KUKA KRL program: EPS_2_25694_AC03A_A_20260223033031.src

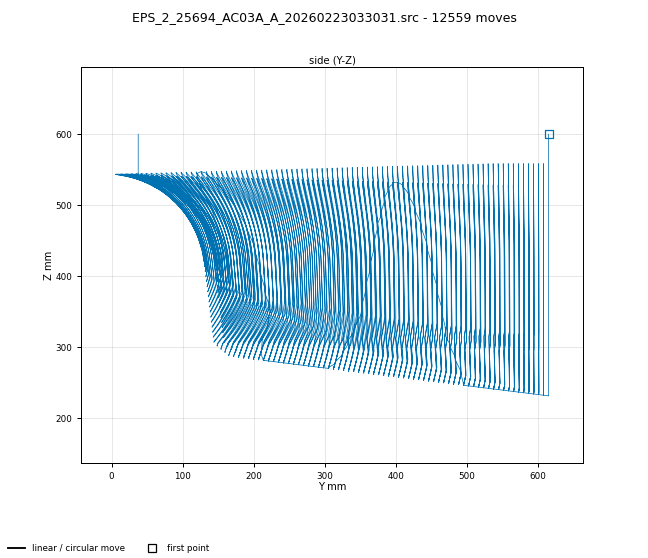
[picture p0: tool path of EPS_2_25694_AC03A_A_20260223033031.src, 12559 of 12561 moves have a stored position in this frame; points joined in program order, loops and branches not executed]
&ACCESS RVP
&REL 4
&COMMENT QRS 19112012
&PARAM EDITMASK = *
DEF PART()
EXT BAS (BAS_COMMAND :IN,REAL :IN )
INT I
BAS (#INITMOV,0 )

;KUKA QRS Post kuka4.cps  Date:22-06-2017 !

File_ID=3050

QRS_PRE_INIT()

;Init var - Until changes are made in qrs_pre_init
Outlet_Square_prg=0
Inlet_1_Square_prg=0
Inlet_2_Square_prg=0
Inlet_3_Square_prg=0
Inlet_4_Square_prg=0
Inlet_5_Square_prg=0

Outlet_1={X 0.000, Y 532.860, Z 433.000, B 0.000, E1 0.000 }
Inlet_1={X 0.000, Y 537.670, Z 428.000, B 0.000, E1 178.000 }
Outlet_1_type=251
Inlet_1_type=201
;QRS#1=Sidecore dimensions
;QRS#2=250-10" PVC SDR 35
;QRS#3=200-8" PVC SDR 35
;QRS#4=
;QRS#5=
;QRS#6=
;QRS#7=
;QRS#8=
;QRS#9=14M PSX
;QRS#10=12-08 PSX
;QRS#11=
;QRS#12=
;QRS#13=
;QRS#14=
;QRS#15=
;QRS#16=1220x127x838 2,75'
;QRS#17=EPS Height
;QRS#18=558,5
;QRS#19=*
;QRS#20= UPDATED VERSION 22-06-2017
;QRS#21=*
Outlet_Square=0100
Inlet_1_Square=0100
Inlet_2_Square=0
Inlet_3_Square=0
Inlet_4_Square=0
Inlet_5_Square=0
Mill_Square=1
Outlet_Square_Prg=205
Inlet_1_Square_prg=204

QRS_INIT()

$ADVANCE=5

; T1
PTP {E1 173.602,E2 173.602}
PTP {X 0,Y 615.5,A -85,B 0,C 180,E1 173.602,E2 173.602,E3 0,E4 0,E5 0,E6 0}
QRS_SPEED_INIT()
LIN {X 0,Y 615.5,Z 600,A -85,B 0,C 180,E1 173.602,E2 173.602,E3 0,E4 0,E5 0,E6 0} C_VEL
LIN {X 0,Y 615.5,Z 241.488,A -85,B 0,C 180,E1 173.602,E2 173.602} C_VEL
LIN {X 0,Y 615.5,Z 233.308,A -85,B 0,C 180,E1 173.602,E2 173.602} C_VEL
LIN {X 0,Y 615.485,Z 231.308,A -85,B 0,C 180,E1 173.415,E2 173.415} C_VEL
LIN {X 0,Y 615.485,Z 231.321,A -85,B 0,C 180,E1 170.801,E2 170.801} C_VEL
LIN {X 0,Y 615.479,Z 231.314,A -85,B 0,C 180,E1 168.139,E2 168.139} C_VEL
LIN {X 0,Y 615.48,Z 231.31,A -85,B 0,C 180,E1 165.45,E2 165.45} C_VEL
LIN {X 0,Y 615.496,Z 231.326,A -85,B 0,C 180,E1 162.729,E2 162.729} C_VEL
LIN {X 0,Y 615.49,Z 231.307,A -85,B 0,C 180,E1 159.967,E2 159.967} C_VEL
LIN {X 0,Y 615.477,Z 231.319,A -85,B 0,C 180,E1 157.155,E2 157.155} C_VEL
LIN {X 0,Y 615.48,Z 231.316,A -85,B 0,C 180,E1 154.431,E2 154.431} C_VEL
LIN {X 0,Y 615.484,Z 231.309,A -85,B 0,C 180,E1 152.084,E2 152.084} C_VEL
LIN {X 0,Y 615.487,Z 231.308,A -85,B 0,C 180,E1 149.839,E2 149.839} C_VEL
LIN {X 0,Y 615.475,Z 231.314,A -85,B 0,C 180,E1 147.541,E2 147.541} C_VEL
LIN {X 0,Y 615.486,Z 231.322,A -85,B 0,C 180,E1 145.184,E2 145.184} C_VEL
LIN {X 0,Y 615.483,Z 231.319,A -85,B 0,C 180,E1 142.757,E2 142.757} C_VEL
LIN {X 0,Y 615.481,Z 231.31,A -85,B 0,C 180,E1 139.911,E2 139.911} C_VEL
LIN {X 0,Y 615.475,Z 231.315,A -85,B 0,C 180,E1 137.645,E2 137.645} C_VEL
LIN {X 0,Y 615.484,Z 231.32,A -85,B 0,C 180,E1 134.931,E2 134.931} C_VEL
LIN {X 0,Y 615.483,Z 231.309,A -85,B 0,C 180,E1 132.079,E2 132.079} C_VEL
LIN {X 0,Y 615.475,Z 231.316,A -85,B 0,C 180,E1 129.75,E2 129.75} C_VEL
LIN {X 0,Y 615.481,Z 231.317,A -85,B 0,C 180,E1 126.935,E2 126.935} C_VEL
LIN {X 0,Y 615.484,Z 231.311,A -85,B 0,C 180,E1 124.699,E2 124.699} C_VEL
LIN {X 0,Y 615.489,Z 231.307,A -85,B 0,C 180,E1 122.33,E2 122.33} C_VEL
LIN {X 0,Y 615.492,Z 231.326,A -85,B 0,C 180,E1 119.406,E2 119.406} C_VEL
LIN {X 0,Y 615.485,Z 231.308,A -85,B 0,C 180,E1 116.444,E2 116.444} C_VEL
LIN {X 0,Y 615.496,Z 231.499,A -85,B 0,C 180,E1 115.424,E2 115.424} C_VEL
LIN {X 0,Y 615.497,Z 234.472,A -85,B 0,C 180,E1 114.991,E2 114.991} C_VEL
LIN {X 0,Y 615.466,Z 256.829,A -85,B 0,C 180,E1 112.137,E2 112.137} C_VEL
LIN {X 0,Y 615.461,Z 277.73,A -85,B 0,C 180,E1 109.512,E2 109.512} C_VEL
LIN {X 0,Y 615.491,Z 299.956,A -85,B 0,C 180,E1 106.757,E2 106.757} C_VEL
LIN {X 0,Y 615.493,Z 315.536,A -85,B 0,C 180,E1 104.866,E2 104.866} C_VEL
LIN {X 0,Y 615.498,Z 318.146,A -85,B 0,C 180,E1 104.802,E2 104.802} C_VEL
LIN {X 0,Y 615.5,Z 424.718,A -85,B 0,C 180,E1 103.537,E2 103.537} C_VEL
LIN {X 0,Y 615.499,Z 437.939,A -85,B 0,C 180,E1 103.243,E2 103.243} C_VEL
LIN {X 0,Y 615.498,Z 450.618,A -85,B 0,C 180,E1 102.823,E2 102.823} C_VEL
LIN {X 0,Y 615.485,Z 462.672,A -85,B 0,C 180,E1 102.279,E2 102.279} C_VEL
LIN {X 0,Y 615.496,Z 474.125,A -85,B 0,C 180,E1 101.61,E2 101.61} C_VEL
LIN {X 0,Y 615.496,Z 484.042,A -85,B 0,C 180,E1 100.889,E2 100.889} C_VEL
LIN {X 0,Y 615.497,Z 493.658,A -85,B 0,C 180,E1 100.028,E2 100.028} C_VEL
LIN {X 0,Y 615.496,Z 502.594,A -85,B 0,C 180,E1 99.033,E2 99.033} C_VEL
LIN {X 0,Y 615.497,Z 509.771,A -85,B 0,C 180,E1 98.041,E2 98.041} C_VEL
LIN {X 0,Y 615.496,Z 516.224,A -85,B 0,C 180,E1 96.898,E2 96.898} C_VEL
LIN {X 0,Y 615.499,Z 520.584,A -85,B 0,C 180,E1 95.898,E2 95.898} C_VEL
LIN {X 0,Y 615.498,Z 522.856,A -85,B 0,C 180,E1 95.241,E2 95.241} C_VEL
LIN {X 0,Y 615.496,Z 524.703,A -85,B 0,C 180,E1 94.584,E2 94.584} C_VEL
LIN {X 0,Y 615.496,Z 526.091,A -85,B 0,C 180,E1 93.928,E2 93.928} C_VEL
LIN {X 0,Y 615.495,Z 527.668,A -85,B 0,C 180,E1 92.618,E2 92.618} C_VEL
LIN {X 0,Y 615.5,Z 527.887,A -85,B 0,C 180,E1 91.963,E2 91.963} C_VEL
LIN {X 0,Y 615.495,Z 527.089,A -85,B 0,C 180,E1 90.654,E2 90.654} C_VEL
LIN {X 0,Y 615.497,Z 526.122,A -85,B 0,C 180,E1 90,E2 90} C_VEL
LIN {X 0,Y 615.494,Z 524.755,A -85,B 0,C 180,E1 89.346,E2 89.346} C_VEL
LIN {X 0,Y 615.496,Z 521.882,A -85,B 0,C 180,E1 88.364,E2 88.364} C_VEL
LIN {X 0,Y 615.498,Z 517.992,A -85,B 0,C 180,E1 87.382,E2 87.382} C_VEL
LIN {X 0,Y 615.496,Z 512.983,A -85,B 0,C 180,E1 86.399,E2 86.399} C_VEL
LIN {X 0,Y 615.498,Z 506.694,A -85,B 0,C 180,E1 85.416,E2 85.416} C_VEL
LIN {X 0,Y 615.498,Z 498.82,A -85,B 0,C 180,E1 84.43,E2 84.43} C_VEL
LIN {X 0,Y 615.498,Z 489.04,A -85,B 0,C 180,E1 83.444,E2 83.444} C_VEL
LIN {X 0,Y 615.499,Z 478.771,A -85,B 0,C 180,E1 82.62,E2 82.62} C_VEL
LIN {X 0,Y 615.488,Z 467.229,A -85,B 0,C 180,E1 81.877,E2 81.877} C_VEL
LIN {X 0,Y 615.497,Z 455.695,A -85,B 0,C 180,E1 81.298,E2 81.298} C_VEL
LIN {X 0,Y 615.498,Z 443.77,A -85,B 0,C 180,E1 80.843,E2 80.843} C_VEL
LIN {X 0,Y 615.499,Z 431.72,A -85,B 0,C 180,E1 80.512,E2 80.512} C_VEL
LIN {X 0,Y 615.497,Z 418.522,A -85,B 0,C 180,E1 80.283,E2 80.283} C_VEL
LIN {X 0,Y 615.49,Z 316.121,A -85,B 0,C 180,E1 79.075,E2 79.075} C_VEL
LIN {X 0,Y 615.49,Z 314.695,A -85,B 0,C 180,E1 78.96,E2 78.96} C_VEL
LIN {X 0,Y 615.492,Z 291.637,A -85,B 0,C 180,E1 76.126,E2 76.126} C_VEL
LIN {X 0,Y 615.485,Z 267.127,A -85,B 0,C 180,E1 73.072,E2 73.072} C_VEL
LIN {X 0,Y 615.462,Z 245.356,A -85,B 0,C 180,E1 70.315,E2 70.315} C_VEL
LIN {X 0,Y 615.495,Z 231.626,A -85,B 0,C 180,E1 68.525,E2 68.525} C_VEL
LIN {X 0,Y 615.481,Z 231.31,A -85,B 0,C 180,E1 67.657,E2 67.657} C_VEL
LIN {X 0,Y 615.478,Z 231.314,A -85,B 0,C 180,E1 65.008,E2 65.008} C_VEL
LIN {X 0,Y 615.482,Z 231.318,A -85,B 0,C 180,E1 62.823,E2 62.823} C_VEL
LIN {X 0,Y 615.477,Z 231.319,A -85,B 0,C 180,E1 60.208,E2 60.208} C_VEL
LIN {X 0,Y 615.493,Z 231.306,A -85,B 0,C 180,E1 57.544,E2 57.544} C_VEL
LIN {X 0,Y 615.48,Z 231.313,A -85,B 0,C 180,E1 55.185,E2 55.185} C_VEL
LIN {X 0,Y 615.485,Z 231.325,A -85,B 0,C 180,E1 52.758,E2 52.758} C_VEL
LIN {X 0,Y 615.48,Z 231.31,A -85,B 0,C 180,E1 49.913,E2 49.913} C_VEL
LIN {X 0,Y 615.496,Z 231.306,A -85,B 0,C 180,E1 47.649,E2 47.649} C_VEL
LIN {X 0,Y 615.486,Z 231.323,A -85,B 0,C 180,E1 44.932,E2 44.932} C_VEL
LIN {X 0,Y 615.481,Z 231.31,A -85,B 0,C 180,E1 42.081,E2 42.081} C_VEL
LIN {X 0,Y 615.49,Z 231.307,A -85,B 0,C 180,E1 39.75,E2 39.75} C_VEL
LIN {X 0,Y 615.486,Z 231.328,A -85,B 0,C 180,E1 36.938,E2 36.938} C_VEL
LIN {X 0,Y 615.487,Z 231.308,A -85,B 0,C 180,E1 34.022,E2 34.022} C_VEL
LIN {X 0,Y 615.482,Z 231.327,A -85,B 0,C 180,E1 31.087,E2 31.087} C_VEL
LIN {X 0,Y 615.477,Z 231.313,A -85,B 0,C 180,E1 28.45,E2 28.45} C_VEL
LIN {X 0,Y 615.481,Z 231.312,A -85,B 0,C 180,E1 25.716,E2 25.716} C_VEL
LIN {X 0,Y 615.478,Z 231.317,A -85,B 0,C 180,E1 23.557,E2 23.557} C_VEL
LIN {X 0,Y 615.483,Z 231.32,A -85,B 0,C 180,E1 21.432,E2 21.432} C_VEL
LIN {X 0,Y 615.476,Z 231.313,A -85,B 0,C 180,E1 18.605,E2 18.605} C_VEL
LIN {X 0,Y 615.478,Z 231.312,A -85,B 0,C 180,E1 15.906,E2 15.906} C_VEL
LIN {X 0,Y 615.491,Z 231.323,A -85,B 0,C 180,E1 13.201,E2 13.201} C_VEL
LIN {X 0,Y 615.485,Z 231.309,A -85,B 0,C 180,E1 10.527,E2 10.527} C_VEL
LIN {X 0,Y 615.479,Z 231.315,A -85,B 0,C 180,E1 7.876,E2 7.876} C_VEL
LIN {X 0,Y 615.485,Z 231.321,A -85,B 0,C 180,E1 5.241,E2 5.241} C_VEL
LIN {X 0,Y 615.487,Z 231.308,A -85,B 0,C 180,E1 2.618,E2 2.618} C_VEL
LIN {X 0,Y 615.479,Z 231.315,A -85,B 0,C 180,E1 0,E2 0} C_VEL
LIN {X 0,Y 615.485,Z 231.321,A -85,B 0,C 180,E1 -2.618,E2 -2.618} C_VEL
LIN {X 0,Y 615.487,Z 231.308,A -85,B 0,C 180,E1 -5.241,E2 -5.241} C_VEL
LIN {X 0,Y 615.479,Z 231.315,A -85,B 0,C 180,E1 -7.876,E2 -7.876} C_VEL
LIN {X 0,Y 615.484,Z 231.321,A -85,B 0,C 180,E1 -10.527,E2 -10.527} C_VEL
LIN {X 0,Y 615.493,Z 231.306,A -85,B 0,C 180,E1 -13.201,E2 -13.201} C_VEL
LIN {X 0,Y 615.482,Z 231.319,A -85,B 0,C 180,E1 -15.905,E2 -15.905} C_VEL
LIN {X 0,Y 615.475,Z 231.316,A -85,B 0,C 180,E1 -18.646,E2 -18.646} C_VEL
LIN {X 0,Y 615.479,Z 231.311,A -85,B 0,C 180,E1 -21.432,E2 -21.432} C_VEL
LIN {X 0,Y 615.483,Z 231.322,A -85,B 0,C 180,E1 -24.272,E2 -24.272} C_VEL
LIN {X 0,Y 615.49,Z 231.307,A -85,B 0,C 180,E1 -27.177,E2 -27.177} C_VEL
LIN {X 0,Y 615.486,Z 231.321,A -85,B 0,C 180,E1 -30.16,E2 -30.16} C_VEL
LIN {X 0,Y 615.472,Z 231.316,A -85,B 0,C 180,E1 -32.458,E2 -32.458} C_VEL
LIN {X 0,Y 615.49,Z 231.307,A -85,B 0,C 180,E1 -34.815,E2 -34.815} C_VEL
LIN {X 0,Y 615.48,Z 231.312,A -85,B 0,C 180,E1 -37.243,E2 -37.243} C_VEL
LIN {X 0,Y 615.482,Z 231.32,A -85,B 0,C 180,E1 -40.09,E2 -40.09} C_VEL
LIN {X 0,Y 615.476,Z 231.314,A -85,B 0,C 180,E1 -42.354,E2 -42.354} C_VEL
LIN {X 0,Y 615.481,Z 231.311,A -85,B 0,C 180,E1 -45.069,E2 -45.069} C_VEL
LIN {X 0,Y 615.484,Z 231.32,A -85,B 0,C 180,E1 -47.92,E2 -47.92} C_VEL
LIN {X 0,Y 615.477,Z 231.313,A -85,B 0,C 180,E1 -50.25,E2 -50.25} C_VEL
LIN {X 0,Y 615.476,Z 231.314,A -85,B 0,C 180,E1 -53.065,E2 -53.065} C_VEL
LIN {X 0,Y 615.482,Z 231.32,A -85,B 0,C 180,E1 -55.3,E2 -55.3} C_VEL
LIN {X 0,Y 615.489,Z 231.322,A -85,B 0,C 180,E1 -57.669,E2 -57.669} C_VEL
LIN {X 0,Y 615.492,Z 231.307,A -85,B 0,C 180,E1 -60.595,E2 -60.595} C_VEL
LIN {X 0,Y 615.485,Z 231.324,A -85,B 0,C 180,E1 -63.556,E2 -63.556} C_VEL
LIN {X 0,Y 615.485,Z 231.308,A -85,B 0,C 180,E1 -66.444,E2 -66.444} C_VEL
LIN {X 0,Y 615.499,Z 231.499,A -85,B 0,C 180,E1 -67.466,E2 -67.466} C_VEL
LIN {X 0,Y 615.496,Z 239.528,A -85,B 0,C 180,E1 -68.393,E2 -68.393} C_VEL
LIN {X 0,Y 615.453,Z 264.946,A -85,B 0,C 180,E1 -71.181,E2 -71.181} C_VEL
LIN {X 0,Y 615.44,Z 287.175,A -85,B 0,C 180,E1 -73.584,E2 -73.584} C_VEL
LIN {X 0,Y 615.491,Z 294.635,A -85,B 0,C 180,E1 -74.371,E2 -74.371} C_VEL
LIN {X 0,Y 615.486,Z 299.642,A -85,B 0,C 180,E1 -74.456,E2 -74.456} C_VEL
LIN {X 0,Y 615.499,Z 433.907,A -85,B 0,C 180,E1 -76.063,E2 -76.063} C_VEL
LIN {X 0,Y 615.497,Z 448.387,A -85,B 0,C 180,E1 -76.379,E2 -76.379} C_VEL
LIN {X 0,Y 615.495,Z 461.695,A -85,B 0,C 180,E1 -76.799,E2 -76.799} C_VEL
LIN {X 0,Y 615.497,Z 473.842,A -85,B 0,C 180,E1 -77.303,E2 -77.303} C_VEL
LIN {X 0,Y 615.484,Z 486.604,A -85,B 0,C 180,E1 -77.972,E2 -77.972} C_VEL
LIN {X 0,Y 615.499,Z 499.343,A -85,B 0,C 180,E1 -78.807,E2 -78.807} C_VEL
LIN {X 0,Y 615.498,Z 509.751,A -85,B 0,C 180,E1 -79.64,E2 -79.64} C_VEL
LIN {X 0,Y 615.496,Z 520.09,A -85,B 0,C 180,E1 -80.636,E2 -80.636} C_VEL
LIN {X 0,Y 615.497,Z 528.604,A -85,B 0,C 180,E1 -81.629,E2 -81.629} C_VEL
LIN {X 0,Y 615.496,Z 536.728,A -85,B 0,C 180,E1 -82.785,E2 -82.785} C_VEL
LIN {X 0,Y 615.497,Z 542.431,A -85,B 0,C 180,E1 -83.773,E2 -83.773} C_VEL
LIN {X 0,Y 615.495,Z 547.081,A -85,B 0,C 180,E1 -84.759,E2 -84.759} C_VEL
LIN {X 0,Y 615.494,Z 551.902,A -85,B 0,C 180,E1 -86.072,E2 -86.072} C_VEL
LIN {X 0,Y 615.496,Z 555.252,A -85,B 0,C 180,E1 -87.382,E2 -87.382} C_VEL
LIN {X 0,Y 615.489,Z 557.229,A -85,B 0,C 180,E1 -88.691,E2 -88.691} C_VEL
LIN {X 0,Y 615.493,Z 557.889,A -85,B 0,C 180,E1 -90,E2 -90} C_VEL
LIN {X 0,Y 615.489,Z 557.229,A -85,B 0,C 180,E1 -91.309,E2 -91.309} C_VEL
LIN {X 0,Y 615.496,Z 555.252,A -85,B 0,C 180,E1 -92.618,E2 -92.618} C_VEL
LIN {X 0,Y 615.494,Z 551.902,A -85,B 0,C 180,E1 -93.928,E2 -93.928} C_VEL
LIN {X 0,Y 615.495,Z 547.08,A -85,B 0,C 180,E1 -95.241,E2 -95.241} C_VEL
LIN {X 0,Y 615.496,Z 540.628,A -85,B 0,C 180,E1 -96.556,E2 -96.556} C_VEL
LIN {X 0,Y 615.496,Z 533.441,A -85,B 0,C 180,E1 -97.71,E2 -97.71} C_VEL
LIN {X 0,Y 615.498,Z 525.904,A -85,B 0,C 180,E1 -98.702,E2 -98.702} C_VEL
LIN {X 0,Y 615.496,Z 516.854,A -85,B 0,C 180,E1 -99.696,E2 -99.696} C_VEL
LIN {X 0,Y 615.498,Z 506.758,A -85,B 0,C 180,E1 -100.618,E2 -100.618} C_VEL
LIN {X 0,Y 615.498,Z 495.859,A -85,B 0,C 180,E1 -101.443,E2 -101.443} C_VEL
LIN {X 0,Y 615.485,Z 483.709,A -85,B 0,C 180,E1 -102.195,E2 -102.195} C_VEL
LIN {X 0,Y 615.494,Z 470.094,A -85,B 0,C 180,E1 -102.865,E2 -102.865} C_VEL
LIN {X 0,Y 615.495,Z 456.839,A -85,B 0,C 180,E1 -103.369,E2 -103.369} C_VEL
LIN {X 0,Y 615.498,Z 443.293,A -85,B 0,C 180,E1 -103.747,E2 -103.747} C_VEL
LIN {X 0,Y 615.498,Z 428.744,A -85,B 0,C 180,E1 -104.013,E2 -104.013} C_VEL
LIN {X 0,Y 615.49,Z 295.04,A -85,B 0,C 180,E1 -105.607,E2 -105.607} C_VEL
LIN {X 0,Y 615.462,Z 289.547,A -85,B 0,C 180,E1 -106.16,E2 -106.16} C_VEL
LIN {X 0,Y 615.445,Z 266.533,A -85,B 0,C 180,E1 -108.647,E2 -108.647} C_VEL
LIN {X 0,Y 615.499,Z 241.116,A -85,B 0,C 180,E1 -111.431,E2 -111.431} C_VEL
LIN {X 0,Y 615.499,Z 231.618,A -85,B 0,C 180,E1 -112.503,E2 -112.503} C_VEL
LIN {X 0,Y 615.483,Z 231.321,A -85,B 0,C 180,E1 -112.844,E2 -112.844} C_VEL
LIN {X 0,Y 615.486,Z 231.308,A -85,B 0,C 180,E1 -115.715,E2 -115.715} C_VEL
LIN {X 0,Y 615.484,Z 231.324,A -85,B 0,C 180,E1 -118.658,E2 -118.658} C_VEL
LIN {X 0,Y 615.479,Z 231.313,A -85,B 0,C 180,E1 -121.085,E2 -121.085} C_VEL
LIN {X 0,Y 615.492,Z 231.306,A -85,B 0,C 180,E1 -123.535,E2 -123.535} C_VEL
LIN {X 0,Y 615.484,Z 231.328,A -85,B 0,C 180,E1 -126.424,E2 -126.424} C_VEL
LIN {X 0,Y 615.482,Z 231.311,A -85,B 0,C 180,E1 -129.061,E2 -129.061} C_VEL
LIN {X 0,Y 615.486,Z 231.308,A -85,B 0,C 180,E1 -131.473,E2 -131.473} C_VEL
LIN {X 0,Y 615.489,Z 231.322,A -85,B 0,C 180,E1 -134.148,E2 -134.148} C_VEL
LIN {X 0,Y 615.482,Z 231.31,A -85,B 0,C 180,E1 -136.952,E2 -136.952} C_VEL
LIN {X 0,Y 615.481,Z 231.31,A -85,B 0,C 180,E1 -139.393,E2 -139.393} C_VEL
LIN {X 0,Y 615.48,Z 231.323,A -85,B 0,C 180,E1 -141.988,E2 -141.988} C_VEL
LIN {X 0,Y 615.479,Z 231.32,A -85,B 0,C 180,E1 -144.384,E2 -144.384} C_VEL
LIN {X 0,Y 615.482,Z 231.311,A -85,B 0,C 180,E1 -146.764,E2 -146.764} C_VEL
LIN {X 0,Y 615.487,Z 231.308,A -85,B 0,C 180,E1 -149.08,E2 -149.08} C_VEL
LIN {X 0,Y 615.477,Z 231.316,A -85,B 0,C 180,E1 -151.55,E2 -151.55} C_VEL
LIN {X 0,Y 615.477,Z 231.319,A -85,B 0,C 180,E1 -154.284,E2 -154.284} C_VEL
LIN {X 0,Y 615.477,Z 231.315,A -85,B 0,C 180,E1 -156.443,E2 -156.443} C_VEL
LIN {X 0,Y 615.479,Z 231.311,A -85,B 0,C 180,E1 -158.568,E2 -158.568} C_VEL
LIN {X 0,Y 615.475,Z 231.316,A -85,B 0,C 180,E1 -161.396,E2 -161.396} C_VEL
LIN {X 0,Y 615.482,Z 231.319,A -85,B 0,C 180,E1 -164.095,E2 -164.095} C_VEL
LIN {X 0,Y 615.493,Z 231.306,A -85,B 0,C 180,E1 -166.799,E2 -166.799} C_VEL
LIN {X 0,Y 615.483,Z 231.32,A -85,B 0,C 180,E1 -169.473,E2 -169.473} C_VEL
LIN {X 0,Y 615.479,Z 231.315,A -85,B 0,C 180,E1 -172.124,E2 -172.124} C_VEL
LIN {X 0,Y 615.487,Z 231.308,A -85,B 0,C 180,E1 -174.759,E2 -174.759} C_VEL
LIN {X 0,Y 615.485,Z 231.321,A -85,B 0,C 180,E1 -177.382,E2 -177.382} C_VEL
LIN {X 0,Y 615.479,Z 231.315,A -85,B 0,C 180,E1 -180,E2 -180} C_VEL
LIN {X 0,Y 615.487,Z 231.308,A -85,B 0,C 180,E1 -182.618,E2 -182.618} C_VEL
LIN {X 0,Y 615.484,Z 231.321,A -85,B 0,C 180,E1 -185.241,E2 -185.241} C_VEL
LIN {X 0,Y 615.485,Z 231.308,A -85,B 0,C 180,E1 -186.585,E2 -186.585} C_VEL
LIN {X 0,Y 614.809,Z 231.468,A -85,B 0,C 180,E1 -187.131,E2 -187.131} C_VEL
LIN {X 0,Y 611.975,Z 231.875,A -85,B 0,C 180,E1 -188.017,E2 -188.017} C_VEL
LIN {X 0,Y 609.583,Z 232.191,A -85,B 0,C 180,E1 -188.729,E2 -188.729} C_VEL
LIN {X 0,Y 608.546,Z 232.311,A -85,B 0,C 180,E1 -189.279,E2 -189.279} C_VEL
LIN {X 0,Y 608.456,Z 232.318,A -85,B 0,C 180,E1 -189.465,E2 -189.465} C_VEL
LIN {X 0,Y 608.455,Z 232.313,A -85,B 0,C 180,E1 -192,E2 -192} C_VEL
LIN {X 0,Y 608.47,Z 232.312,A -85,B 0,C 180,E1 -194.721,E2 -194.721} C_VEL
LIN {X 0,Y 608.457,Z 232.319,A -85,B 0,C 180,E1 -197.477,E2 -197.477} C_VEL
LIN {X 0,Y 608.46,Z 232.311,A -85,B 0,C 180,E1 -200.275,E2 -200.275} C_VEL
LIN {X 0,Y 608.452,Z 232.313,A -85,B 0,C 180,E1 -202.477,E2 -202.477} C_VEL
LIN {X 0,Y 608.453,Z 232.314,A -85,B 0,C 180,E1 -204.571,E2 -204.571} C_VEL
LIN {X 0,Y 608.482,Z 232.317,A -85,B 0,C 180,E1 -207.21,E2 -207.21} C_VEL
LIN {X 0,Y 608.467,Z 232.31,A -85,B 0,C 180,E1 -209.973,E2 -209.973} C_VEL
LIN {X 0,Y 608.451,Z 232.315,A -85,B 0,C 180,E1 -212.522,E2 -212.522} C_VEL
LIN {X 0,Y 608.441,Z 232.319,A -85,B 0,C 180,E1 -215.278,E2 -215.278} C_VEL
LIN {X 0,Y 608.466,Z 232.311,A -85,B 0,C 180,E1 -217.747,E2 -217.747} C_VEL
LIN {X 0,Y 608.445,Z 232.315,A -85,B 0,C 180,E1 -220.329,E2 -220.329} C_VEL
LIN {X 0,Y 608.452,Z 232.321,A -85,B 0,C 180,E1 -222.961,E2 -222.961} C_VEL
LIN {X 0,Y 608.459,Z 232.312,A -85,B 0,C 180,E1 -225.737,E2 -225.737} C_VEL
LIN {X 0,Y 608.46,Z 232.32,A -85,B 0,C 180,E1 -228.659,E2 -228.659} C_VEL
LIN {X 0,Y 608.462,Z 232.311,A -85,B 0,C 180,E1 -231.761,E2 -231.761} C_VEL
LIN {X 0,Y 608.445,Z 232.314,A -85,B 0,C 180,E1 -233.956,E2 -233.956} C_VEL
LIN {X 0,Y 608.446,Z 232.318,A -85,B 0,C 180,E1 -236.329,E2 -236.329} C_VEL
LIN {X 0,Y 608.448,Z 232.321,A -85,B 0,C 180,E1 -238.733,E2 -238.733} C_VEL
LIN {X 0,Y 608.474,Z 232.31,A -85,B 0,C 180,E1 -241.381,E2 -241.381} C_VEL
LIN {X 0,Y 608.473,Z 232.318,A -85,B 0,C 180,E1 -244.28,E2 -244.28} C_VEL
LIN {X 0,Y 608.531,Z 232.698,A -85,B 0,C 180,E1 -244.484,E2 -244.484} C_VEL
LIN {X 0,Y 608.565,Z 248.251,A -85,B 0,C 180,E1 -246.521,E2 -246.521} C_VEL
LIN {X 0,Y 608.534,Z 270.042,A -85,B 0,C 180,E1 -249.306,E2 -249.306} C_VEL
LIN {X 0,Y 608.506,Z 292.884,A -85,B 0,C 180,E1 -252.178,E2 -252.178} C_VEL
LIN {X 0,Y 608.484,Z 315.353,A -85,B 0,C 180,E1 -254.959,E2 -254.959} C_VEL
LIN {X 0,Y 608.564,Z 316.492,A -85,B 0,C 180,E1 -255.025,E2 -255.025} C_VEL
LIN {X 0,Y 608.551,Z 424.72,A -85,B 0,C 180,E1 -256.327,E2 -256.327} C_VEL
LIN {X 0,Y 608.548,Z 437.979,A -85,B 0,C 180,E1 -256.624,E2 -256.624} C_VEL
LIN {X 0,Y 608.527,Z 450.13,A -85,B 0,C 180,E1 -257.027,E2 -257.027} C_VEL
LIN {X 0,Y 608.491,Z 462.397,A -85,B 0,C 180,E1 -257.578,E2 -257.578} C_VEL
LIN {X 0,Y 608.501,Z 473.977,A -85,B 0,C 180,E1 -258.255,E2 -258.255} C_VEL
LIN {X 0,Y 608.481,Z 484.737,A -85,B 0,C 180,E1 -259.042,E2 -259.042} C_VEL
LIN {X 0,Y 608.482,Z 493.745,A -85,B 0,C 180,E1 -259.855,E2 -259.855} C_VEL
LIN {X 0,Y 608.47,Z 502.779,A -85,B 0,C 180,E1 -260.862,E2 -260.862} C_VEL
LIN {X 0,Y 608.463,Z 510.05,A -85,B 0,C 180,E1 -261.866,E2 -261.866} C_VEL
LIN {X 0,Y 608.445,Z 514.948,A -85,B 0,C 180,E1 -262.7,E2 -262.7} C_VEL
LIN {X 0,Y 608.452,Z 519.411,A -85,B 0,C 180,E1 -263.632,E2 -263.632} C_VEL
LIN {X 0,Y 608.442,Z 523.341,A -85,B 0,C 180,E1 -264.698,E2 -264.698} C_VEL
LIN {X 0,Y 608.429,Z 525.219,A -85,B 0,C 180,E1 -265.362,E2 -265.362} C_VEL
LIN {X 0,Y 608.433,Z 526.646,A -85,B 0,C 180,E1 -266.026,E2 -266.026} C_VEL
LIN {X 0,Y 608.421,Z 528.261,A -85,B 0,C 180,E1 -267.352,E2 -267.352} C_VEL
LIN {X 0,Y 608.445,Z 528.498,A -85,B 0,C 180,E1 -268.014,E2 -268.014} C_VEL
LIN {X 0,Y 608.447,Z 528.305,A -85,B 0,C 180,E1 -268.676,E2 -268.676} C_VEL
LIN {X 0,Y 608.437,Z 526.753,A -85,B 0,C 180,E1 -270,E2 -270} C_VEL
LIN {X 0,Y 608.437,Z 525.387,A -85,B 0,C 180,E1 -270.662,E2 -270.662} C_VEL
LIN {X 0,Y 608.44,Z 522.503,A -85,B 0,C 180,E1 -271.655,E2 -271.655} C_VEL
LIN {X 0,Y 608.432,Z 518.599,A -85,B 0,C 180,E1 -272.648,E2 -272.648} C_VEL
LIN {X 0,Y 608.449,Z 513.569,A -85,B 0,C 180,E1 -273.642,E2 -273.642} C_VEL
LIN {X 0,Y 608.465,Z 507.261,A -85,B 0,C 180,E1 -274.637,E2 -274.637} C_VEL
LIN {X 0,Y 608.47,Z 499.369,A -85,B 0,C 180,E1 -275.634,E2 -275.634} C_VEL
LIN {X 0,Y 608.485,Z 489.571,A -85,B 0,C 180,E1 -276.632,E2 -276.632} C_VEL
LIN {X 0,Y 608.479,Z 479.318,A -85,B 0,C 180,E1 -277.466,E2 -277.466} C_VEL
LIN {X 0,Y 608.505,Z 467.794,A -85,B 0,C 180,E1 -278.217,E2 -278.217} C_VEL
LIN {X 0,Y 608.519,Z 456.378,A -85,B 0,C 180,E1 -278.802,E2 -278.802} C_VEL
LIN {X 0,Y 608.547,Z 444.602,A -85,B 0,C 180,E1 -279.263,E2 -279.263} C_VEL
LIN {X 0,Y 608.549,Z 431.929,A -85,B 0,C 180,E1 -279.619,E2 -279.619} C_VEL
LIN {X 0,Y 608.565,Z 418.82,A -85,B 0,C 180,E1 -279.849,E2 -279.849} C_VEL
LIN {X 0,Y 608.549,Z 316.322,A -85,B 0,C 180,E1 -281.069,E2 -281.069} C_VEL
LIN {X 0,Y 608.478,Z 314.814,A -85,B 0,C 180,E1 -281.193,E2 -281.193} C_VEL
LIN {X 0,Y 608.504,Z 291.888,A -85,B 0,C 180,E1 -284.036,E2 -284.036} C_VEL
LIN {X 0,Y 608.55,Z 268.697,A -85,B 0,C 180,E1 -286.954,E2 -286.954} C_VEL
LIN {X 0,Y 608.553,Z 246.913,A -85,B 0,C 180,E1 -289.742,E2 -289.742} C_VEL
LIN {X 0,Y 608.534,Z 232.74,A -85,B 0,C 180,E1 -291.6,E2 -291.6} C_VEL
LIN {X 0,Y 608.479,Z 232.409,A -85,B 0,C 180,E1 -291.691,E2 -291.691} C_VEL
LIN {X 0,Y 608.448,Z 232.313,A -85,B 0,C 180,E1 -294.571,E2 -294.571} C_VEL
LIN {X 0,Y 608.476,Z 232.315,A -85,B 0,C 180,E1 -297.206,E2 -297.206} C_VEL
LIN {X 0,Y 608.46,Z 232.314,A -85,B 0,C 180,E1 -299.969,E2 -299.969} C_VEL
LIN {X 0,Y 608.462,Z 232.314,A -85,B 0,C 180,E1 -302.879,E2 -302.879} C_VEL
LIN {X 0,Y 608.439,Z 232.323,A -85,B 0,C 180,E1 -305.277,E2 -305.277} C_VEL
LIN {X 0,Y 608.464,Z 232.315,A -85,B 0,C 180,E1 -307.746,E2 -307.746} C_VEL
LIN {X 0,Y 608.447,Z 232.313,A -85,B 0,C 180,E1 -310.328,E2 -310.328} C_VEL
LIN {X 0,Y 608.485,Z 232.318,A -85,B 0,C 180,E1 -313.31,E2 -313.31} C_VEL
LIN {X 0,Y 608.467,Z 232.311,A -85,B 0,C 180,E1 -316.13,E2 -316.13} C_VEL
LIN {X 0,Y 608.453,Z 232.317,A -85,B 0,C 180,E1 -318.823,E2 -318.823} C_VEL
LIN {X 0,Y 608.471,Z 232.315,A -85,B 0,C 180,E1 -321.412,E2 -321.412} C_VEL
LIN {X 0,Y 608.476,Z 232.31,A -85,B 0,C 180,E1 -323.949,E2 -323.949} C_VEL
LIN {X 0,Y 608.46,Z 232.312,A -85,B 0,C 180,E1 -326.329,E2 -326.329} C_VEL
LIN {X 0,Y 608.473,Z 232.316,A -85,B 0,C 180,E1 -328.727,E2 -328.727} C_VEL
LIN {X 0,Y 608.465,Z 232.314,A -85,B 0,C 180,E1 -331.38,E2 -331.38} C_VEL
LIN {X 0,Y 608.438,Z 232.314,A -85,B 0,C 180,E1 -333.964,E2 -333.964} C_VEL
LIN {X 0,Y 608.466,Z 232.312,A -85,B 0,C 180,E1 -336.155,E2 -336.155} C_VEL
LIN {X 0,Y 608.469,Z 232.313,A -85,B 0,C 180,E1 -338.308,E2 -338.308} C_VEL
LIN {X 0,Y 608.462,Z 232.314,A -85,B 0,C 180,E1 -341.284,E2 -341.284} C_VEL
LIN {X 0,Y 608.455,Z 232.312,A -85,B 0,C 180,E1 -343.906,E2 -343.906} C_VEL
LIN {X 0,Y 608.465,Z 232.321,A -85,B 0,C 180,E1 -346.643,E2 -346.643} C_VEL
LIN {X 0,Y 608.459,Z 232.312,A -85,B 0,C 180,E1 -349.35,E2 -349.35} C_VEL
LIN {X 0,Y 608.47,Z 232.312,A -85,B 0,C 180,E1 -352.033,E2 -352.033} C_VEL
LIN {X 0,Y 608.463,Z 232.319,A -85,B 0,C 180,E1 -354.698,E2 -354.698} C_VEL
LIN {X 0,Y 608.478,Z 232.31,A -85,B 0,C 180,E1 -357.352,E2 -357.352} C_VEL
LIN {X 0,Y 608.469,Z 232.313,A -85,B 0,C 180,E1 -360,E2 -360} C_VEL
LIN {X 0,Y 608.476,Z 232.316,A -85,B 0,C 180,E1 -362.648,E2 -362.648} C_VEL
LIN {X 0,Y 608.465,Z 232.311,A -85,B 0,C 180,E1 -365.302,E2 -365.302} C_VEL
LIN {X 0,Y 608.471,Z 232.314,A -85,B 0,C 180,E1 -367.967,E2 -367.967} C_VEL
LIN {X 0,Y 608.46,Z 232.316,A -85,B 0,C 180,E1 -370.65,E2 -370.65} C_VEL
LIN {X 0,Y 608.467,Z 232.311,A -85,B 0,C 180,E1 -373.356,E2 -373.356} C_VEL
LIN {X 0,Y 608.457,Z 232.32,A -85,B 0,C 180,E1 -376.094,E2 -376.094} C_VEL
LIN {X 0,Y 608.449,Z 232.314,A -85,B 0,C 180,E1 -378.87,E2 -378.87} C_VEL
LIN {X 0,Y 608.467,Z 232.314,A -85,B 0,C 180,E1 -381.691,E2 -381.691} C_VEL
LIN {X 0,Y 608.453,Z 232.315,A -85,B 0,C 180,E1 -384.571,E2 -384.571} C_VEL
LIN {X 0,Y 608.482,Z 232.309,A -85,B 0,C 180,E1 -387.21,E2 -387.21} C_VEL
LIN {X 0,Y 608.467,Z 232.321,A -85,B 0,C 180,E1 -389.973,E2 -389.973} C_VEL
LIN {X 0,Y 608.449,Z 232.315,A -85,B 0,C 180,E1 -392.522,E2 -392.522} C_VEL
LIN {X 0,Y 608.441,Z 232.315,A -85,B 0,C 180,E1 -395.278,E2 -395.278} C_VEL
LIN {X 0,Y 608.466,Z 232.319,A -85,B 0,C 180,E1 -397.746,E2 -397.746} C_VEL
LIN {X 0,Y 608.447,Z 232.316,A -85,B 0,C 180,E1 -400.33,E2 -400.33} C_VEL
LIN {X 0,Y 608.448,Z 232.313,A -85,B 0,C 180,E1 -402.96,E2 -402.96} C_VEL
LIN {X 0,Y 608.457,Z 232.322,A -85,B 0,C 180,E1 -405.736,E2 -405.736} C_VEL
LIN {X 0,Y 608.462,Z 232.311,A -85,B 0,C 180,E1 -408.658,E2 -408.658} C_VEL
LIN {X 0,Y 608.462,Z 232.319,A -85,B 0,C 180,E1 -411.76,E2 -411.76} C_VEL
LIN {X 0,Y 608.443,Z 232.318,A -85,B 0,C 180,E1 -413.955,E2 -413.955} C_VEL
LIN {X 0,Y 608.465,Z 232.311,A -85,B 0,C 180,E1 -416.33,E2 -416.33} C_VEL
LIN {X 0,Y 608.445,Z 232.314,A -85,B 0,C 180,E1 -418.733,E2 -418.733} C_VEL
LIN {X 0,Y 608.472,Z 232.319,A -85,B 0,C 180,E1 -421.38,E2 -421.38} C_VEL
LIN {X 0,Y 608.475,Z 232.31,A -85,B 0,C 180,E1 -424.279,E2 -424.279} C_VEL
LIN {X 0,Y 608.449,Z 232.317,A -85,B 0,C 180,E1 -426.876,E2 -426.876} C_VEL
LIN {X 0,Y 608.509,Z 232.559,A -85,B 0,C 180,E1 -427.337,E2 -427.337} C_VEL
LIN {X 0,Y 608.606,Z 245.883,A -85,B 0,C 180,E1 -428.847,E2 -428.847} C_VEL
LIN {X 0,Y 608.534,Z 268.922,A -85,B 0,C 180,E1 -431.396,E2 -431.396} C_VEL
LIN {X 0,Y 608.534,Z 294.637,A -85,B 0,C 180,E1 -434.188,E2 -434.188} C_VEL
LIN {X 0,Y 608.668,Z 297.853,A -85,B 0,C 180,E1 -434.256,E2 -434.256} C_VEL
LIN {X 0,Y 608.621,Z 432.926,A -85,B 0,C 180,E1 -435.885,E2 -435.885} C_VEL
LIN {X 0,Y 608.607,Z 446.871,A -85,B 0,C 180,E1 -436.179,E2 -436.179} C_VEL
LIN {X 0,Y 608.565,Z 460.595,A -85,B 0,C 180,E1 -436.604,E2 -436.604} C_VEL
LIN {X 0,Y 608.562,Z 473.888,A -85,B 0,C 180,E1 -437.156,E2 -437.156} C_VEL
LIN {X 0,Y 608.513,Z 486.684,A -85,B 0,C 180,E1 -437.832,E2 -437.832} C_VEL
LIN {X 0,Y 608.499,Z 499.474,A -85,B 0,C 180,E1 -438.677,E2 -438.677} C_VEL
LIN {X 0,Y 608.496,Z 509.933,A -85,B 0,C 180,E1 -439.519,E2 -439.519} C_VEL
LIN {X 0,Y 608.479,Z 520.336,A -85,B 0,C 180,E1 -440.527,E2 -440.527} C_VEL
LIN {X 0,Y 608.464,Z 528.915,A -85,B 0,C 180,E1 -441.532,E2 -441.532} C_VEL
LIN {X 0,Y 608.461,Z 537.114,A -85,B 0,C 180,E1 -442.701,E2 -442.701} C_VEL
LIN {X 0,Y 608.444,Z 543.545,A -85,B 0,C 180,E1 -443.831,E2 -443.831} C_VEL
LIN {X 0,Y 608.437,Z 548.962,A -85,B 0,C 180,E1 -445.03,E2 -445.03} C_VEL
LIN {X 0,Y 608.431,Z 552.442,A -85,B 0,C 180,E1 -446.026,E2 -446.026} C_VEL
LIN {X 0,Y 608.424,Z 555.831,A -85,B 0,C 180,E1 -447.352,E2 -447.352} C_VEL
LIN {X 0,Y 608.442,Z 557.83,A -85,B 0,C 180,E1 -448.676,E2 -448.676} C_VEL
LIN {X 0,Y 608.433,Z 558.5,A -85,B 0,C 180,E1 -450,E2 -450} C_VEL
LIN {X 0,Y 608.442,Z 557.83,A -85,B 0,C 180,E1 -451.324,E2 -451.324} C_VEL
LIN {X 0,Y 608.424,Z 555.831,A -85,B 0,C 180,E1 -452.648,E2 -452.648} C_VEL
LIN {X 0,Y 608.431,Z 552.441,A -85,B 0,C 180,E1 -453.974,E2 -453.974} C_VEL
LIN {X 0,Y 608.44,Z 547.568,A -85,B 0,C 180,E1 -455.302,E2 -455.302} C_VEL
LIN {X 0,Y 608.445,Z 541.211,A -85,B 0,C 180,E1 -456.603,E2 -456.603} C_VEL
LIN {X 0,Y 608.453,Z 533.798,A -85,B 0,C 180,E1 -457.8,E2 -457.8} C_VEL
LIN {X 0,Y 608.473,Z 524.824,A -85,B 0,C 180,E1 -458.97,E2 -458.97} C_VEL
LIN {X 0,Y 608.473,Z 515.392,A -85,B 0,C 180,E1 -459.977,E2 -459.977} C_VEL
LIN {X 0,Y 608.506,Z 504.046,A -85,B 0,C 180,E1 -460.973,E2 -460.973} C_VEL
LIN {X 0,Y 608.531,Z 492.15,A -85,B 0,C 180,E1 -461.829,E2 -461.829} C_VEL
LIN {X 0,Y 608.529,Z 479.075,A -85,B 0,C 180,E1 -462.591,E2 -462.591} C_VEL
LIN {X 0,Y 608.561,Z 466.176,A -85,B 0,C 180,E1 -463.184,E2 -463.184} C_VEL
LIN {X 0,Y 608.597,Z 452.187,A -85,B 0,C 180,E1 -463.672,E2 -463.672} C_VEL
LIN {X 0,Y 608.621,Z 438.461,A -85,B 0,C 180,E1 -464.012,E2 -464.012} C_VEL
LIN {X 0,Y 608.626,Z 422.178,A -85,B 0,C 180,E1 -464.257,E2 -464.257} C_VEL
LIN {X 0,Y 608.577,Z 295.047,A -85,B 0,C 180,E1 -465.789,E2 -465.789} C_VEL
LIN {X 0,Y 608.488,Z 285.601,A -85,B 0,C 180,E1 -466.783,E2 -466.783} C_VEL
LIN {X 0,Y 608.594,Z 260.181,A -85,B 0,C 180,E1 -469.566,E2 -469.566} C_VEL
LIN {X 0,Y 608.642,Z 234.761,A -85,B 0,C 180,E1 -472.398,E2 -472.398} C_VEL
LIN {X 0,Y 608.477,Z 232.45,A -85,B 0,C 180,E1 -472.689,E2 -472.689} C_VEL
LIN {X 0,Y 608.453,Z 232.314,A -85,B 0,C 180,E1 -475.3,E2 -475.3} C_VEL
LIN {X 0,Y 608.443,Z 232.314,A -85,B 0,C 180,E1 -477.518,E2 -477.518} C_VEL
LIN {X 0,Y 608.459,Z 232.314,A -85,B 0,C 180,E1 -479.97,E2 -479.97} C_VEL
LIN {X 0,Y 608.459,Z 232.315,A -85,B 0,C 180,E1 -482.879,E2 -482.879} C_VEL
LIN {X 0,Y 608.44,Z 232.314,A -85,B 0,C 180,E1 -485.277,E2 -485.277} C_VEL
LIN {X 0,Y 608.464,Z 232.312,A -85,B 0,C 180,E1 -487.746,E2 -487.746} C_VEL
LIN {X 0,Y 608.447,Z 232.324,A -85,B 0,C 180,E1 -490.328,E2 -490.328} C_VEL
LIN {X 0,Y 608.482,Z 232.309,A -85,B 0,C 180,E1 -493.31,E2 -493.31} C_VEL
LIN {X 0,Y 608.466,Z 232.319,A -85,B 0,C 180,E1 -496.13,E2 -496.13} C_VEL
LIN {X 0,Y 608.452,Z 232.314,A -85,B 0,C 180,E1 -498.823,E2 -498.823} C_VEL
LIN {X 0,Y 608.468,Z 232.311,A -85,B 0,C 180,E1 -501.412,E2 -501.412} C_VEL
LIN {X 0,Y 608.474,Z 232.317,A -85,B 0,C 180,E1 -503.95,E2 -503.95} C_VEL
LIN {X 0,Y 608.459,Z 232.318,A -85,B 0,C 180,E1 -506.329,E2 -506.329} C_VEL
LIN {X 0,Y 608.472,Z 232.311,A -85,B 0,C 180,E1 -508.727,E2 -508.727} C_VEL
LIN {X 0,Y 608.465,Z 232.312,A -85,B 0,C 180,E1 -511.38,E2 -511.38} C_VEL
LIN {X 0,Y 608.437,Z 232.325,A -85,B 0,C 180,E1 -513.964,E2 -513.964} C_VEL
LIN {X 0,Y 608.469,Z 232.317,A -85,B 0,C 180,E1 -516.155,E2 -516.155} C_VEL
LIN {X 0,Y 608.468,Z 232.314,A -85,B 0,C 180,E1 -518.309,E2 -518.309} C_VEL
LIN {X 0,Y 608.461,Z 232.313,A -85,B 0,C 180,E1 -521.284,E2 -521.284} C_VEL
LIN {X 0,Y 608.457,Z 232.321,A -85,B 0,C 180,E1 -523.906,E2 -523.906} C_VEL
LIN {X 0,Y 608.467,Z 232.311,A -85,B 0,C 180,E1 -526.644,E2 -526.644} C_VEL
LIN {X 0,Y 608.459,Z 232.316,A -85,B 0,C 180,E1 -529.35,E2 -529.35} C_VEL
LIN {X 0,Y 608.471,Z 232.314,A -85,B 0,C 180,E1 -532.033,E2 -532.033} C_VEL
LIN {X 0,Y 608.465,Z 232.311,A -85,B 0,C 180,E1 -534.698,E2 -534.698} C_VEL
LIN {X 0,Y 608.475,Z 232.316,A -85,B 0,C 180,E1 -537.352,E2 -537.352} C_VEL
LIN {X 0,Y 608.47,Z 232.313,A -85,B 0,C 180,E1 -540,E2 -540} C_VEL
LIN {X 0,Y 608.477,Z 232.309,A -85,B 0,C 180,E1 -542.648,E2 -542.648} C_VEL
LIN {X 0,Y 608.463,Z 232.319,A -85,B 0,C 180,E1 -545.302,E2 -545.302} C_VEL
LIN {X 0,Y 608.47,Z 232.312,A -85,B 0,C 180,E1 -547.967,E2 -547.967} C_VEL
LIN {X 0,Y 608.456,Z 232.318,A -85,B 0,C 180,E1 -549.465,E2 -549.465} C_VEL
LIN {X 0,Y 607.774,Z 232.399,A -85,B 0,C 180,E1 -550.018,E2 -550.018} C_VEL
LIN {X 0,Y 604.918,Z 232.756,A -85,B 0,C 180,E1 -550.915,E2 -550.915} C_VEL
LIN {X 0,Y 602.516,Z 233.057,A -85,B 0,C 180,E1 -551.636,E2 -551.636} C_VEL
LIN {X 0,Y 601.488,Z 233.181,A -85,B 0,C 180,E1 -552.193,E2 -552.193} C_VEL
LIN {X 0,Y 601.405,Z 233.19,A -85,B 0,C 180,E1 -552.381,E2 -552.381} C_VEL
LIN {X 0,Y 601.425,Z 233.192,A -85,B 0,C 180,E1 -554.897,E2 -554.897} C_VEL
LIN {X 0,Y 601.429,Z 233.193,A -85,B 0,C 180,E1 -556.986,E2 -556.986} C_VEL
LIN {X 0,Y 601.407,Z 233.192,A -85,B 0,C 180,E1 -559.81,E2 -559.81} C_VEL
LIN {X 0,Y 601.406,Z 233.193,A -85,B 0,C 180,E1 -562.684,E2 -562.684} C_VEL
LIN {X 0,Y 601.401,Z 233.197,A -85,B 0,C 180,E1 -564.879,E2 -564.879} C_VEL
LIN {X 0,Y 601.417,Z 233.189,A -85,B 0,C 180,E1 -567.868,E2 -567.868} C_VEL
LIN {X 0,Y 601.425,Z 233.188,A -85,B 0,C 180,E1 -570.165,E2 -570.165} C_VEL
LIN {X 0,Y 601.414,Z 233.195,A -85,B 0,C 180,E1 -572.716,E2 -572.716} C_VEL
LIN {X 0,Y 601.409,Z 233.198,A -85,B 0,C 180,E1 -575.115,E2 -575.115} C_VEL
LIN {X 0,Y 601.433,Z 233.19,A -85,B 0,C 180,E1 -577.42,E2 -577.42} C_VEL
LIN {X 0,Y 601.41,Z 233.189,A -85,B 0,C 180,E1 -579.996,E2 -579.996} C_VEL
LIN {X 0,Y 601.408,Z 233.197,A -85,B 0,C 180,E1 -582.671,E2 -582.671} C_VEL
LIN {X 0,Y 601.425,Z 233.189,A -85,B 0,C 180,E1 -585.483,E2 -585.483} C_VEL
LIN {X 0,Y 601.423,Z 233.192,A -85,B 0,C 180,E1 -588.408,E2 -588.408} C_VEL
LIN {X 0,Y 601.43,Z 233.186,A -85,B 0,C 180,E1 -591.53,E2 -591.53} C_VEL
LIN {X 0,Y 601.386,Z 233.197,A -85,B 0,C 180,E1 -594.246,E2 -594.246} C_VEL
LIN {X 0,Y 601.42,Z 233.199,A -85,B 0,C 180,E1 -596.687,E2 -596.687} C_VEL
LIN {X 0,Y 601.413,Z 233.193,A -85,B 0,C 180,E1 -599.058,E2 -599.058} C_VEL
LIN {X 0,Y 601.433,Z 233.187,A -85,B 0,C 180,E1 -601.374,E2 -601.374} C_VEL
LIN {X 0,Y 601.452,Z 233.265,A -85,B 0,C 180,E1 -604.203,E2 -604.203} C_VEL
LIN {X 0,Y 601.581,Z 234.071,A -85,B 0,C 180,E1 -604.39,E2 -604.39} C_VEL
LIN {X 0,Y 601.724,Z 245.256,A -85,B 0,C 180,E1 -605.871,E2 -605.871} C_VEL
LIN {X 0,Y 601.615,Z 267.6,A -85,B 0,C 180,E1 -608.769,E2 -608.769} C_VEL
LIN {X 0,Y 601.52,Z 289.902,A -85,B 0,C 180,E1 -611.612,E2 -611.612} C_VEL
LIN {X 0,Y 601.483,Z 312.165,A -85,B 0,C 180,E1 -614.411,E2 -614.411} C_VEL
LIN {X 0,Y 601.478,Z 315.835,A -85,B 0,C 180,E1 -614.845,E2 -614.845} C_VEL
LIN {X 0,Y 601.679,Z 321.424,A -85,B 0,C 180,E1 -614.936,E2 -614.936} C_VEL
LIN {X 0,Y 601.61,Z 424.406,A -85,B 0,C 180,E1 -616.184,E2 -616.184} C_VEL
LIN {X 0,Y 601.586,Z 437.901,A -85,B 0,C 180,E1 -616.488,E2 -616.488} C_VEL
LIN {X 0,Y 601.542,Z 450.637,A -85,B 0,C 180,E1 -616.917,E2 -616.917} C_VEL
LIN {X 0,Y 601.5,Z 461.952,A -85,B 0,C 180,E1 -617.431,E2 -617.431} C_VEL
LIN {X 0,Y 601.481,Z 473.624,A -85,B 0,C 180,E1 -618.116,E2 -618.116} C_VEL
LIN {X 0,Y 601.448,Z 483.494,A -85,B 0,C 180,E1 -618.836,E2 -618.836} C_VEL
LIN {X 0,Y 601.419,Z 493.518,A -85,B 0,C 180,E1 -619.735,E2 -619.735} C_VEL
LIN {X 0,Y 601.405,Z 502.59,A -85,B 0,C 180,E1 -620.754,E2 -620.754} C_VEL
LIN {X 0,Y 601.383,Z 509.894,A -85,B 0,C 180,E1 -621.769,E2 -621.769} C_VEL
LIN {X 0,Y 601.352,Z 514.823,A -85,B 0,C 180,E1 -622.614,E2 -622.614} C_VEL
LIN {X 0,Y 601.356,Z 519.526,A -85,B 0,C 180,E1 -623.607,E2 -623.607} C_VEL
LIN {X 0,Y 601.353,Z 523.268,A -85,B 0,C 180,E1 -624.635,E2 -624.635} C_VEL
LIN {X 0,Y 601.329,Z 525.158,A -85,B 0,C 180,E1 -625.307,E2 -625.307} C_VEL
LIN {X 0,Y 601.343,Z 526.607,A -85,B 0,C 180,E1 -625.979,E2 -625.979} C_VEL
LIN {X 0,Y 601.32,Z 528.246,A -85,B 0,C 180,E1 -627.32,E2 -627.32} C_VEL
LIN {X 0,Y 601.343,Z 528.494,A -85,B 0,C 180,E1 -627.991,E2 -627.991} C_VEL
LIN {X 0,Y 601.347,Z 528.321,A -85,B 0,C 180,E1 -628.661,E2 -628.661} C_VEL
LIN {X 0,Y 601.338,Z 526.791,A -85,B 0,C 180,E1 -630,E2 -630} C_VEL
LIN {X 0,Y 601.338,Z 525.439,A -85,B 0,C 180,E1 -630.67,E2 -630.67} C_VEL
LIN {X 0,Y 601.359,Z 522.576,A -85,B 0,C 180,E1 -631.674,E2 -631.674} C_VEL
LIN {X 0,Y 601.337,Z 518.697,A -85,B 0,C 180,E1 -632.679,E2 -632.679} C_VEL
LIN {X 0,Y 601.368,Z 513.694,A -85,B 0,C 180,E1 -633.685,E2 -633.685} C_VEL
LIN {X 0,Y 601.401,Z 507.421,A -85,B 0,C 180,E1 -634.692,E2 -634.692} C_VEL
LIN {X 0,Y 601.399,Z 499.574,A -85,B 0,C 180,E1 -635.701,E2 -635.701} C_VEL
LIN {X 0,Y 601.437,Z 489.816,A -85,B 0,C 180,E1 -636.71,E2 -636.71} C_VEL
LIN {X 0,Y 601.457,Z 479.64,A -85,B 0,C 180,E1 -637.554,E2 -637.554} C_VEL
LIN {X 0,Y 601.513,Z 468.184,A -85,B 0,C 180,E1 -638.313,E2 -638.313} C_VEL
LIN {X 0,Y 601.539,Z 456.889,A -85,B 0,C 180,E1 -638.905,E2 -638.905} C_VEL
LIN {X 0,Y 601.582,Z 445.313,A -85,B 0,C 180,E1 -639.371,E2 -639.371} C_VEL
LIN {X 0,Y 601.594,Z 432.025,A -85,B 0,C 180,E1 -639.752,E2 -639.752} C_VEL
LIN {X 0,Y 601.641,Z 418.969,A -85,B 0,C 180,E1 -639.985,E2 -639.985} C_VEL
LIN {X 0,Y 601.541,Z 316.396,A -85,B 0,C 180,E1 -641.221,E2 -641.221} C_VEL
LIN {X 0,Y 601.466,Z 315.325,A -85,B 0,C 180,E1 -641.29,E2 -641.29} C_VEL
LIN {X 0,Y 601.531,Z 292.645,A -85,B 0,C 180,E1 -644.131,E2 -644.131} C_VEL
LIN {X 0,Y 601.628,Z 267.528,A -85,B 0,C 180,E1 -647.33,E2 -647.33} C_VEL
LIN {X 0,Y 601.707,Z 244.388,A -85,B 0,C 180,E1 -650.333,E2 -650.333} C_VEL
LIN {X 0,Y 601.735,Z 234.873,A -85,B 0,C 180,E1 -651.586,E2 -651.586} C_VEL
LIN {X 0,Y 601.453,Z 233.287,A -85,B 0,C 180,E1 -651.867,E2 -651.867} C_VEL
LIN {X 0,Y 601.431,Z 233.188,A -85,B 0,C 180,E1 -654.29,E2 -654.29} C_VEL
LIN {X 0,Y 601.449,Z 233.188,A -85,B 0,C 180,E1 -657.111,E2 -657.111} C_VEL
LIN {X 0,Y 601.419,Z 233.199,A -85,B 0,C 180,E1 -659.393,E2 -659.393} C_VEL
LIN {X 0,Y 601.403,Z 233.196,A -85,B 0,C 180,E1 -661.726,E2 -661.726} C_VEL
LIN {X 0,Y 601.428,Z 233.188,A -85,B 0,C 180,E1 -664.118,E2 -664.118} C_VEL
LIN {X 0,Y 601.435,Z 233.197,A -85,B 0,C 180,E1 -667.381,E2 -667.381} C_VEL
LIN {X 0,Y 601.4,Z 233.192,A -85,B 0,C 180,E1 -669.995,E2 -669.995} C_VEL
LIN {X 0,Y 601.414,Z 233.191,A -85,B 0,C 180,E1 -672.669,E2 -672.669} C_VEL
LIN {X 0,Y 601.425,Z 233.193,A -85,B 0,C 180,E1 -675.481,E2 -675.481} C_VEL
LIN {X 0,Y 601.421,Z 233.189,A -85,B 0,C 180,E1 -678.406,E2 -678.406} C_VEL
LIN {X 0,Y 601.436,Z 233.192,A -85,B 0,C 180,E1 -680.875,E2 -680.875} C_VEL
LIN {X 0,Y 601.441,Z 233.187,A -85,B 0,C 180,E1 -683.733,E2 -683.733} C_VEL
LIN {X 0,Y 601.422,Z 233.192,A -85,B 0,C 180,E1 -686.686,E2 -686.686} C_VEL
LIN {X 0,Y 601.428,Z 233.197,A -85,B 0,C 180,E1 -689.058,E2 -689.058} C_VEL
LIN {X 0,Y 601.425,Z 233.191,A -85,B 0,C 180,E1 -691.372,E2 -691.372} C_VEL
LIN {X 0,Y 601.399,Z 233.192,A -85,B 0,C 180,E1 -693.636,E2 -693.636} C_VEL
LIN {X 0,Y 601.416,Z 233.195,A -85,B 0,C 180,E1 -696.589,E2 -696.589} C_VEL
LIN {X 0,Y 601.424,Z 233.189,A -85,B 0,C 180,E1 -699.478,E2 -699.478} C_VEL
LIN {X 0,Y 601.398,Z 233.195,A -85,B 0,C 180,E1 -702.311,E2 -702.311} C_VEL
LIN {X 0,Y 601.412,Z 233.194,A -85,B 0,C 180,E1 -704.408,E2 -704.408} C_VEL
LIN {X 0,Y 601.42,Z 233.191,A -85,B 0,C 180,E1 -707.172,E2 -707.172} C_VEL
LIN {X 0,Y 601.427,Z 233.188,A -85,B 0,C 180,E1 -709.905,E2 -709.905} C_VEL
LIN {X 0,Y 601.448,Z 233.195,A -85,B 0,C 180,E1 -712.615,E2 -712.615} C_VEL
LIN {X 0,Y 601.422,Z 233.188,A -85,B 0,C 180,E1 -715.308,E2 -715.308} C_VEL
LIN {X 0,Y 601.419,Z 233.191,A -85,B 0,C 180,E1 -717.991,E2 -717.991} C_VEL
LIN {X 0,Y 601.448,Z 233.192,A -85,B 0,C 180,E1 -720.669,E2 -720.669} C_VEL
LIN {X 0,Y 601.427,Z 233.188,A -85,B 0,C 180,E1 -723.349,E2 -723.349} C_VEL
LIN {X 0,Y 601.406,Z 233.195,A -85,B 0,C 180,E1 -726.037,E2 -726.037} C_VEL
LIN {X 0,Y 601.433,Z 233.191,A -85,B 0,C 180,E1 -728.737,E2 -728.737} C_VEL
LIN {X 0,Y 601.429,Z 233.187,A -85,B 0,C 180,E1 -731.458,E2 -731.458} C_VEL
LIN {X 0,Y 601.411,Z 233.2,A -85,B 0,C 180,E1 -734.205,E2 -734.205} C_VEL
LIN {X 0,Y 601.428,Z 233.188,A -85,B 0,C 180,E1 -736.986,E2 -736.986} C_VEL
LIN {X 0,Y 601.406,Z 233.195,A -85,B 0,C 180,E1 -739.809,E2 -739.809} C_VEL
LIN {X 0,Y 601.404,Z 233.192,A -85,B 0,C 180,E1 -742.683,E2 -742.683} C_VEL
LIN {X 0,Y 601.4,Z 233.191,A -85,B 0,C 180,E1 -744.879,E2 -744.879} C_VEL
LIN {X 0,Y 601.417,Z 233.197,A -85,B 0,C 180,E1 -747.867,E2 -747.867} C_VEL
LIN {X 0,Y 601.442,Z 233.192,A -85,B 0,C 180,E1 -750.163,E2 -750.163} C_VEL
LIN {X 0,Y 601.412,Z 233.19,A -85,B 0,C 180,E1 -752.716,E2 -752.716} C_VEL
LIN {X 0,Y 601.41,Z 233.19,A -85,B 0,C 180,E1 -755.115,E2 -755.115} C_VEL
LIN {X 0,Y 601.43,Z 233.19,A -85,B 0,C 180,E1 -757.419,E2 -757.419} C_VEL
LIN {X 0,Y 601.407,Z 233.197,A -85,B 0,C 180,E1 -759.995,E2 -759.995} C_VEL
LIN {X 0,Y 601.406,Z 233.19,A -85,B 0,C 180,E1 -762.671,E2 -762.671} C_VEL
LIN {X 0,Y 601.421,Z 233.195,A -85,B 0,C 180,E1 -765.483,E2 -765.483} C_VEL
LIN {X 0,Y 601.423,Z 233.187,A -85,B 0,C 180,E1 -768.407,E2 -768.407} C_VEL
LIN {X 0,Y 601.428,Z 233.196,A -85,B 0,C 180,E1 -771.53,E2 -771.53} C_VEL
LIN {X 0,Y 601.385,Z 233.193,A -85,B 0,C 180,E1 -774.246,E2 -774.246} C_VEL
LIN {X 0,Y 601.428,Z 233.188,A -85,B 0,C 180,E1 -776.687,E2 -776.687} C_VEL
LIN {X 0,Y 601.41,Z 233.192,A -85,B 0,C 180,E1 -779.058,E2 -779.058} C_VEL
LIN {X 0,Y 601.432,Z 233.196,A -85,B 0,C 180,E1 -781.374,E2 -781.374} C_VEL
LIN {X 0,Y 601.414,Z 233.191,A -85,B 0,C 180,E1 -784.133,E2 -784.133} C_VEL
LIN {X 0,Y 601.418,Z 233.193,A -85,B 0,C 180,E1 -786.59,E2 -786.59} C_VEL
LIN {X 0,Y 601.458,Z 233.433,A -85,B 0,C 180,E1 -787.156,E2 -787.156} C_VEL
LIN {X 0,Y 601.807,Z 236.899,A -85,B 0,C 180,E1 -787.577,E2 -787.577} C_VEL
LIN {X 0,Y 601.668,Z 263.359,A -85,B 0,C 180,E1 -790.555,E2 -790.555} C_VEL
LIN {X 0,Y 601.527,Z 287.12,A -85,B 0,C 180,E1 -793.184,E2 -793.184} C_VEL
LIN {X 0,Y 601.619,Z 295.04,A -85,B 0,C 180,E1 -794.023,E2 -794.023} C_VEL
LIN {X 0,Y 601.848,Z 301.43,A -85,B 0,C 180,E1 -794.116,E2 -794.116} C_VEL
LIN {X 0,Y 601.739,Z 433.912,A -85,B 0,C 180,E1 -795.738,E2 -795.738} C_VEL
LIN {X 0,Y 601.688,Z 448.487,A -85,B 0,C 180,E1 -796.063,E2 -796.063} C_VEL
LIN {X 0,Y 601.667,Z 462.841,A -85,B 0,C 180,E1 -796.533,E2 -796.533} C_VEL
LIN {X 0,Y 601.606,Z 475.639,A -85,B 0,C 180,E1 -797.09,E2 -797.09} C_VEL
LIN {X 0,Y 601.544,Z 488.098,A -85,B 0,C 180,E1 -797.775,E2 -797.775} C_VEL
LIN {X 0,Y 601.504,Z 499.476,A -85,B 0,C 180,E1 -798.543,E2 -798.543} C_VEL
LIN {X 0,Y 601.482,Z 509.934,A -85,B 0,C 180,E1 -799.396,E2 -799.396} C_VEL
LIN {X 0,Y 601.43,Z 520.336,A -85,B 0,C 180,E1 -800.415,E2 -800.415} C_VEL
LIN {X 0,Y 601.407,Z 528.915,A -85,B 0,C 180,E1 -801.431,E2 -801.431} C_VEL
LIN {X 0,Y 601.392,Z 537.115,A -85,B 0,C 180,E1 -802.614,E2 -802.614} C_VEL
LIN {X 0,Y 601.361,Z 542.75,A -85,B 0,C 180,E1 -803.604,E2 -803.604} C_VEL
LIN {X 0,Y 601.355,Z 547.568,A -85,B 0,C 180,E1 -804.635,E2 -804.635} C_VEL
LIN {X 0,Y 601.343,Z 552.442,A -85,B 0,C 180,E1 -805.979,E2 -805.979} C_VEL
LIN {X 0,Y 601.324,Z 555.831,A -85,B 0,C 180,E1 -807.321,E2 -807.321} C_VEL
LIN {X 0,Y 601.342,Z 557.831,A -85,B 0,C 180,E1 -808.661,E2 -808.661} C_VEL
LIN {X 0,Y 601.333,Z 558.5,A -85,B 0,C 180,E1 -810,E2 -810} C_VEL
LIN {X 0,Y 601.342,Z 557.831,A -85,B 0,C 180,E1 -811.339,E2 -811.339} C_VEL
LIN {X 0,Y 601.324,Z 555.832,A -85,B 0,C 180,E1 -812.68,E2 -812.68} C_VEL
LIN {X 0,Y 601.343,Z 552.442,A -85,B 0,C 180,E1 -814.021,E2 -814.021} C_VEL
LIN {X 0,Y 601.355,Z 547.568,A -85,B 0,C 180,E1 -815.365,E2 -815.365} C_VEL
LIN {X 0,Y 601.372,Z 541.623,A -85,B 0,C 180,E1 -816.605,E2 -816.605} C_VEL
LIN {X 0,Y 601.386,Z 534.919,A -85,B 0,C 180,E1 -817.723,E2 -817.723} C_VEL
LIN {X 0,Y 601.412,Z 526.199,A -85,B 0,C 180,E1 -818.907,E2 -818.907} C_VEL
LIN {X 0,Y 601.433,Z 517.083,A -85,B 0,C 180,E1 -819.925,E2 -819.925} C_VEL
LIN {X 0,Y 601.497,Z 506.827,A -85,B 0,C 180,E1 -820.877,E2 -820.877} C_VEL
LIN {X 0,Y 601.533,Z 495.972,A -85,B 0,C 180,E1 -821.712,E2 -821.712} C_VEL
LIN {X 0,Y 601.575,Z 483.78,A -85,B 0,C 180,E1 -822.482,E2 -822.482} C_VEL
LIN {X 0,Y 601.628,Z 472.097,A -85,B 0,C 180,E1 -823.081,E2 -823.081} C_VEL
LIN {X 0,Y 601.669,Z 458.942,A -85,B 0,C 180,E1 -823.613,E2 -823.613} C_VEL
LIN {X 0,Y 601.706,Z 445.033,A -85,B 0,C 180,E1 -824.028,E2 -824.028} C_VEL
LIN {X 0,Y 601.732,Z 430.558,A -85,B 0,C 180,E1 -824.314,E2 -824.314} C_VEL
LIN {X 0,Y 601.708,Z 295.66,A -85,B 0,C 180,E1 -825.959,E2 -825.959} C_VEL
LIN {X 0,Y 601.551,Z 294.375,A -85,B 0,C 180,E1 -826.022,E2 -826.022} C_VEL
LIN {X 0,Y 601.61,Z 269.673,A -85,B 0,C 180,E1 -828.743,E2 -828.743} C_VEL
LIN {X 0,Y 601.747,Z 245.882,A -85,B 0,C 180,E1 -831.406,E2 -831.406} C_VEL
LIN {X 0,Y 601.735,Z 234.689,A -85,B 0,C 180,E1 -832.678,E2 -832.678} C_VEL
LIN {X 0,Y 601.423,Z 233.257,A -85,B 0,C 180,E1 -832.895,E2 -832.895} C_VEL
LIN {X 0,Y 601.436,Z 233.187,A -85,B 0,C 180,E1 -835.617,E2 -835.617} C_VEL
LIN {X 0,Y 601.402,Z 233.192,A -85,B 0,C 180,E1 -837.868,E2 -837.868} C_VEL
LIN {X 0,Y 601.426,Z 233.193,A -85,B 0,C 180,E1 -840.164,E2 -840.164} C_VEL
LIN {X 0,Y 601.425,Z 233.194,A -85,B 0,C 180,E1 -842.716,E2 -842.716} C_VEL
LIN {X 0,Y 601.394,Z 233.192,A -85,B 0,C 180,E1 -845.112,E2 -845.112} C_VEL
LIN {X 0,Y 601.432,Z 233.186,A -85,B 0,C 180,E1 -847.419,E2 -847.419} C_VEL
LIN {X 0,Y 601.398,Z 233.196,A -85,B 0,C 180,E1 -849.995,E2 -849.995} C_VEL
LIN {X 0,Y 601.413,Z 233.194,A -85,B 0,C 180,E1 -852.669,E2 -852.669} C_VEL
LIN {X 0,Y 601.422,Z 233.189,A -85,B 0,C 180,E1 -855.482,E2 -855.482} C_VEL
LIN {X 0,Y 601.42,Z 233.195,A -85,B 0,C 180,E1 -858.406,E2 -858.406} C_VEL
LIN {X 0,Y 601.434,Z 233.188,A -85,B 0,C 180,E1 -860.875,E2 -860.875} C_VEL
LIN {X 0,Y 601.439,Z 233.19,A -85,B 0,C 180,E1 -863.733,E2 -863.733} C_VEL
LIN {X 0,Y 601.428,Z 233.198,A -85,B 0,C 180,E1 -866.064,E2 -866.064} C_VEL
LIN {X 0,Y 601.427,Z 233.187,A -85,B 0,C 180,E1 -869.059,E2 -869.059} C_VEL
LIN {X 0,Y 601.425,Z 233.189,A -85,B 0,C 180,E1 -871.373,E2 -871.373} C_VEL
LIN {X 0,Y 601.399,Z 233.196,A -85,B 0,C 180,E1 -873.636,E2 -873.636} C_VEL
LIN {X 0,Y 601.417,Z 233.19,A -85,B 0,C 180,E1 -876.59,E2 -876.59} C_VEL
LIN {X 0,Y 601.424,Z 233.192,A -85,B 0,C 180,E1 -879.478,E2 -879.478} C_VEL
LIN {X 0,Y 601.397,Z 233.194,A -85,B 0,C 180,E1 -882.312,E2 -882.312} C_VEL
LIN {X 0,Y 601.414,Z 233.191,A -85,B 0,C 180,E1 -884.409,E2 -884.409} C_VEL
LIN {X 0,Y 601.419,Z 233.19,A -85,B 0,C 180,E1 -887.172,E2 -887.172} C_VEL
LIN {X 0,Y 601.427,Z 233.195,A -85,B 0,C 180,E1 -889.905,E2 -889.905} C_VEL
LIN {X 0,Y 601.447,Z 233.185,A -85,B 0,C 180,E1 -892.615,E2 -892.615} C_VEL
LIN {X 0,Y 601.42,Z 233.194,A -85,B 0,C 180,E1 -895.308,E2 -895.308} C_VEL
LIN {X 0,Y 601.42,Z 233.192,A -85,B 0,C 180,E1 -897.991,E2 -897.991} C_VEL
LIN {X 0,Y 601.446,Z 233.185,A -85,B 0,C 180,E1 -900.67,E2 -900.67} C_VEL
LIN {X 0,Y 601.428,Z 233.195,A -85,B 0,C 180,E1 -903.35,E2 -903.35} C_VEL
LIN {X 0,Y 601.407,Z 233.192,A -85,B 0,C 180,E1 -906.037,E2 -906.037} C_VEL
LIN {X 0,Y 601.433,Z 233.188,A -85,B 0,C 180,E1 -908.738,E2 -908.738} C_VEL
LIN {X 0,Y 601.43,Z 233.196,A -85,B 0,C 180,E1 -911.459,E2 -911.459} C_VEL
LIN {X 0,Y 601.405,Z 233.19,A -85,B 0,C 180,E1 -912.381,E2 -912.381} C_VEL
LIN {X 0,Y 600.742,Z 233.278,A -85,B 0,C 180,E1 -912.941,E2 -912.941} C_VEL
LIN {X 0,Y 597.892,Z 233.634,A -85,B 0,C 180,E1 -913.848,E2 -913.848} C_VEL
LIN {X 0,Y 595.48,Z 233.936,A -85,B 0,C 180,E1 -914.578,E2 -914.578} C_VEL
LIN {X 0,Y 594.442,Z 234.065,A -85,B 0,C 180,E1 -915.142,E2 -915.142} C_VEL
LIN {X 0,Y 594.357,Z 234.072,A -85,B 0,C 180,E1 -915.333,E2 -915.333} C_VEL
LIN {X 0,Y 594.376,Z 234.067,A -85,B 0,C 180,E1 -917.905,E2 -917.905} C_VEL
LIN {X 0,Y 594.372,Z 234.072,A -85,B 0,C 180,E1 -920.917,E2 -920.917} C_VEL
LIN {X 0,Y 594.388,Z 234.066,A -85,B 0,C 180,E1 -923.704,E2 -923.704} C_VEL
LIN {X 0,Y 594.384,Z 234.069,A -85,B 0,C 180,E1 -926.7,E2 -926.7} C_VEL
LIN {X 0,Y 594.376,Z 234.074,A -85,B 0,C 180,E1 -928.999,E2 -928.999} C_VEL
LIN {X 0,Y 594.388,Z 234.066,A -85,B 0,C 180,E1 -931.646,E2 -931.646} C_VEL
LIN {X 0,Y 594.391,Z 234.067,A -85,B 0,C 180,E1 -934.58,E2 -934.58} C_VEL
LIN {X 0,Y 594.384,Z 234.073,A -85,B 0,C 180,E1 -937.087,E2 -937.087} C_VEL
LIN {X 0,Y 594.375,Z 234.065,A -85,B 0,C 180,E1 -939.775,E2 -939.775} C_VEL
LIN {X 0,Y 594.365,Z 234.07,A -85,B 0,C 180,E1 -942.376,E2 -942.376} C_VEL
LIN {X 0,Y 594.363,Z 234.072,A -85,B 0,C 180,E1 -945.192,E2 -945.192} C_VEL
LIN {X 0,Y 594.371,Z 234.066,A -85,B 0,C 180,E1 -947.626,E2 -947.626} C_VEL
LIN {X 0,Y 594.372,Z 234.071,A -85,B 0,C 180,E1 -950.32,E2 -950.32} C_VEL
LIN {X 0,Y 594.383,Z 234.072,A -85,B 0,C 180,E1 -952.914,E2 -952.914} C_VEL
LIN {X 0,Y 594.372,Z 234.066,A -85,B 0,C 180,E1 -955.864,E2 -955.864} C_VEL
LIN {X 0,Y 594.371,Z 234.075,A -85,B 0,C 180,E1 -958.65,E2 -958.65} C_VEL
LIN {X 0,Y 594.386,Z 234.068,A -85,B 0,C 180,E1 -961.043,E2 -961.043} C_VEL
LIN {X 0,Y 594.399,Z 234.182,A -85,B 0,C 180,E1 -964.057,E2 -964.057} C_VEL
LIN {X 0,Y 594.831,Z 236.659,A -85,B 0,C 180,E1 -964.453,E2 -964.453} C_VEL
LIN {X 0,Y 594.753,Z 256.233,A -85,B 0,C 180,E1 -967.049,E2 -967.049} C_VEL
LIN {X 0,Y 594.625,Z 277.165,A -85,B 0,C 180,E1 -969.775,E2 -969.775} C_VEL
LIN {X 0,Y 594.505,Z 299.451,A -85,B 0,C 180,E1 -972.633,E2 -972.633} C_VEL
LIN {X 0,Y 594.452,Z 315.811,A -85,B 0,C 180,E1 -974.683,E2 -974.683} C_VEL
LIN {X 0,Y 594.77,Z 319.435,A -85,B 0,C 180,E1 -974.757,E2 -974.757} C_VEL
LIN {X 0,Y 594.681,Z 424.544,A -85,B 0,C 180,E1 -976.046,E2 -976.046} C_VEL
LIN {X 0,Y 594.618,Z 437.823,A -85,B 0,C 180,E1 -976.349,E2 -976.349} C_VEL
LIN {X 0,Y 594.603,Z 450.017,A -85,B 0,C 180,E1 -976.762,E2 -976.762} C_VEL
LIN {X 0,Y 594.505,Z 461.488,A -85,B 0,C 180,E1 -977.281,E2 -977.281} C_VEL
LIN {X 0,Y 594.472,Z 473.27,A -85,B 0,C 180,E1 -977.973,E2 -977.973} C_VEL
LIN {X 0,Y 594.414,Z 484.065,A -85,B 0,C 180,E1 -978.772,E2 -978.772} C_VEL
LIN {X 0,Y 594.379,Z 493.287,A -85,B 0,C 180,E1 -979.612,E2 -979.612} C_VEL
LIN {X 0,Y 594.315,Z 502.401,A -85,B 0,C 180,E1 -980.642,E2 -980.642} C_VEL
LIN {X 0,Y 594.287,Z 509.738,A -85,B 0,C 180,E1 -981.671,E2 -981.671} C_VEL
LIN {X 0,Y 594.281,Z 514.697,A -85,B 0,C 180,E1 -982.526,E2 -982.526} C_VEL
LIN {X 0,Y 594.274,Z 518.96,A -85,B 0,C 180,E1 -983.418,E2 -983.418} C_VEL
LIN {X 0,Y 594.271,Z 523.196,A -85,B 0,C 180,E1 -984.571,E2 -984.571} C_VEL
LIN {X 0,Y 594.229,Z 525.098,A -85,B 0,C 180,E1 -985.251,E2 -985.251} C_VEL
LIN {X 0,Y 594.255,Z 526.568,A -85,B 0,C 180,E1 -985.931,E2 -985.931} C_VEL
LIN {X 0,Y 594.259,Z 527.594,A -85,B 0,C 180,E1 -986.61,E2 -986.61} C_VEL
LIN {X 0,Y 594.242,Z 528.488,A -85,B 0,C 180,E1 -987.967,E2 -987.967} C_VEL
LIN {X 0,Y 594.247,Z 528.338,A -85,B 0,C 180,E1 -988.645,E2 -988.645} C_VEL
LIN {X 0,Y 594.238,Z 526.83,A -85,B 0,C 180,E1 -990,E2 -990} C_VEL
LIN {X 0,Y 594.239,Z 525.489,A -85,B 0,C 180,E1 -990.678,E2 -990.678} C_VEL
LIN {X 0,Y 594.28,Z 522.648,A -85,B 0,C 180,E1 -991.694,E2 -991.694} C_VEL
LIN {X 0,Y 594.243,Z 518.795,A -85,B 0,C 180,E1 -992.711,E2 -992.711} C_VEL
LIN {X 0,Y 594.289,Z 513.819,A -85,B 0,C 180,E1 -993.729,E2 -993.729} C_VEL
LIN {X 0,Y 594.339,Z 507.577,A -85,B 0,C 180,E1 -994.748,E2 -994.748} C_VEL
LIN {X 0,Y 594.33,Z 499.78,A -85,B 0,C 180,E1 -995.769,E2 -995.769} C_VEL
LIN {X 0,Y 594.393,Z 490.061,A -85,B 0,C 180,E1 -996.79,E2 -996.79} C_VEL
LIN {X 0,Y 594.436,Z 479.961,A -85,B 0,C 180,E1 -997.643,E2 -997.643} C_VEL
LIN {X 0,Y 594.518,Z 468.574,A -85,B 0,C 180,E1 -998.412,E2 -998.412} C_VEL
LIN {X 0,Y 594.553,Z 457.375,A -85,B 0,C 180,E1 -999.011,E2 -999.011} C_VEL
LIN {X 0,Y 594.624,Z 446.003,A -85,B 0,C 180,E1 -999.481,E2 -999.481} C_VEL
LIN {X 0,Y 594.668,Z 433.024,A -85,B 0,C 180,E1 -999.867,E2 -999.867} C_VEL
LIN {X 0,Y 594.675,Z 420.625,A -85,B 0,C 180,E1 -1000.103,E2 -1000.103} C_VEL
LIN {X 0,Y 594.709,Z 317.743,A -85,B 0,C 180,E1 -1001.355,E2 -1001.355} C_VEL
LIN {X 0,Y 594.464,Z 315.815,A -85,B 0,C 180,E1 -1001.406,E2 -1001.406} C_VEL
LIN {X 0,Y 594.557,Z 294.459,A -85,B 0,C 180,E1 -1004.093,E2 -1004.093} C_VEL
LIN {X 0,Y 594.657,Z 270.449,A -85,B 0,C 180,E1 -1007.185,E2 -1007.185} C_VEL
LIN {X 0,Y 594.763,Z 250.025,A -85,B 0,C 180,E1 -1009.86,E2 -1009.86} C_VEL
LIN {X 0,Y 594.833,Z 236.431,A -85,B 0,C 180,E1 -1011.667,E2 -1011.667} C_VEL
LIN {X 0,Y 594.379,Z 234.167,A -85,B 0,C 180,E1 -1012.05,E2 -1012.05} C_VEL
LIN {X 0,Y 594.392,Z 234.064,A -85,B 0,C 180,E1 -1014.445,E2 -1014.445} C_VEL
LIN {X 0,Y 594.384,Z 234.064,A -85,B 0,C 180,E1 -1016.699,E2 -1016.699} C_VEL
LIN {X 0,Y 594.384,Z 234.069,A -85,B 0,C 180,E1 -1018.998,E2 -1018.998} C_VEL
LIN {X 0,Y 594.379,Z 234.072,A -85,B 0,C 180,E1 -1021.642,E2 -1021.642} C_VEL
LIN {X 0,Y 594.379,Z 234.065,A -85,B 0,C 180,E1 -1024.579,E2 -1024.579} C_VEL
LIN {X 0,Y 594.389,Z 234.07,A -85,B 0,C 180,E1 -1027.607,E2 -1027.607} C_VEL
LIN {X 0,Y 594.367,Z 234.068,A -85,B 0,C 180,E1 -1030.566,E2 -1030.566} C_VEL
LIN {X 0,Y 594.38,Z 234.075,A -85,B 0,C 180,E1 -1033.297,E2 -1033.297} C_VEL
LIN {X 0,Y 594.366,Z 234.067,A -85,B 0,C 180,E1 -1036.16,E2 -1036.16} C_VEL
LIN {X 0,Y 594.375,Z 234.075,A -85,B 0,C 180,E1 -1039.177,E2 -1039.177} C_VEL
LIN {X 0,Y 594.384,Z 234.065,A -85,B 0,C 180,E1 -1042.059,E2 -1042.059} C_VEL
LIN {X 0,Y 594.381,Z 234.069,A -85,B 0,C 180,E1 -1044.671,E2 -1044.671} C_VEL
LIN {X 0,Y 594.373,Z 234.075,A -85,B 0,C 180,E1 -1047.088,E2 -1047.088} C_VEL
LIN {X 0,Y 594.397,Z 234.064,A -85,B 0,C 180,E1 -1049.668,E2 -1049.668} C_VEL
LIN {X 0,Y 594.387,Z 234.068,A -85,B 0,C 180,E1 -1052.539,E2 -1052.539} C_VEL
LIN {X 0,Y 594.373,Z 234.076,A -85,B 0,C 180,E1 -1054.806,E2 -1054.806} C_VEL
LIN {X 0,Y 594.358,Z 234.072,A -85,B 0,C 180,E1 -1057.264,E2 -1057.264} C_VEL
LIN {X 0,Y 594.373,Z 234.066,A -85,B 0,C 180,E1 -1059.946,E2 -1059.946} C_VEL
LIN {X 0,Y 594.387,Z 234.074,A -85,B 0,C 180,E1 -1062.806,E2 -1062.806} C_VEL
LIN {X 0,Y 594.382,Z 234.065,A -85,B 0,C 180,E1 -1065.825,E2 -1065.825} C_VEL
LIN {X 0,Y 594.388,Z 234.071,A -85,B 0,C 180,E1 -1068.404,E2 -1068.404} C_VEL
LIN {X 0,Y 594.394,Z 234.066,A -85,B 0,C 180,E1 -1071.158,E2 -1071.158} C_VEL
LIN {X 0,Y 594.363,Z 234.069,A -85,B 0,C 180,E1 -1073.891,E2 -1073.891} C_VEL
LIN {X 0,Y 594.38,Z 234.075,A -85,B 0,C 180,E1 -1076.61,E2 -1076.61} C_VEL
LIN {X 0,Y 594.417,Z 234.061,A -85,B 0,C 180,E1 -1079.322,E2 -1079.322} C_VEL
LIN {X 0,Y 594.389,Z 234.068,A -85,B 0,C 180,E1 -1082.033,E2 -1082.033} C_VEL
LIN {X 0,Y 594.389,Z 234.068,A -85,B 0,C 180,E1 -1084.747,E2 -1084.747} C_VEL
LIN {X 0,Y 594.395,Z 234.064,A -85,B 0,C 180,E1 -1087.473,E2 -1087.473} C_VEL
LIN {X 0,Y 594.387,Z 234.074,A -85,B 0,C 180,E1 -1090.216,E2 -1090.216} C_VEL
LIN {X 0,Y 594.367,Z 234.068,A -85,B 0,C 180,E1 -1092.983,E2 -1092.983} C_VEL
LIN {X 0,Y 594.366,Z 234.07,A -85,B 0,C 180,E1 -1095.781,E2 -1095.781} C_VEL
LIN {X 0,Y 594.378,Z 234.069,A -85,B 0,C 180,E1 -1098.618,E2 -1098.618} C_VEL
LIN {X 0,Y 594.362,Z 234.069,A -85,B 0,C 180,E1 -1101.503,E2 -1101.503} C_VEL
LIN {X 0,Y 594.382,Z 234.069,A -85,B 0,C 180,E1 -1104.446,E2 -1104.446} C_VEL
LIN {X 0,Y 594.384,Z 234.066,A -85,B 0,C 180,E1 -1106.699,E2 -1106.699} C_VEL
LIN {X 0,Y 594.375,Z 234.065,A -85,B 0,C 180,E1 -1108.999,E2 -1108.999} C_VEL
LIN {X 0,Y 594.385,Z 234.069,A -85,B 0,C 180,E1 -1111.646,E2 -1111.646} C_VEL
LIN {X 0,Y 594.392,Z 234.065,A -85,B 0,C 180,E1 -1114.579,E2 -1114.579} C_VEL
LIN {X 0,Y 594.382,Z 234.064,A -85,B 0,C 180,E1 -1117.087,E2 -1117.087} C_VEL
LIN {X 0,Y 594.373,Z 234.076,A -85,B 0,C 180,E1 -1119.775,E2 -1119.775} C_VEL
LIN {X 0,Y 594.363,Z 234.069,A -85,B 0,C 180,E1 -1122.376,E2 -1122.376} C_VEL
LIN {X 0,Y 594.359,Z 234.071,A -85,B 0,C 180,E1 -1125.192,E2 -1125.192} C_VEL
LIN {X 0,Y 594.37,Z 234.075,A -85,B 0,C 180,E1 -1127.626,E2 -1127.626} C_VEL
LIN {X 0,Y 594.37,Z 234.068,A -85,B 0,C 180,E1 -1130.32,E2 -1130.32} C_VEL
LIN {X 0,Y 594.379,Z 234.067,A -85,B 0,C 180,E1 -1132.914,E2 -1132.914} C_VEL
LIN {X 0,Y 594.38,Z 234.071,A -85,B 0,C 180,E1 -1135.862,E2 -1135.862} C_VEL
LIN {X 0,Y 594.376,Z 234.065,A -85,B 0,C 180,E1 -1138.651,E2 -1138.651} C_VEL
LIN {X 0,Y 594.383,Z 234.069,A -85,B 0,C 180,E1 -1141.042,E2 -1141.042} C_VEL
LIN {X 0,Y 594.388,Z 234.068,A -85,B 0,C 180,E1 -1143.977,E2 -1143.977} C_VEL
LIN {X 0,Y 594.385,Z 234.072,A -85,B 0,C 180,E1 -1146.666,E2 -1146.666} C_VEL
LIN {X 0,Y 594.422,Z 234.282,A -85,B 0,C 180,E1 -1146.967,E2 -1146.967} C_VEL
LIN {X 0,Y 594.954,Z 238.475,A -85,B 0,C 180,E1 -1147.486,E2 -1147.486} C_VEL
LIN {X 0,Y 594.764,Z 264.948,A -85,B 0,C 180,E1 -1150.5,E2 -1150.5} C_VEL
LIN {X 0,Y 594.575,Z 289.29,A -85,B 0,C 180,E1 -1153.224,E2 -1153.224} C_VEL
LIN {X 0,Y 594.64,Z 295.039,A -85,B 0,C 180,E1 -1153.831,E2 -1153.831} C_VEL
LIN {X 0,Y 595.014,Z 299.642,A -85,B 0,C 180,E1 -1153.907,E2 -1153.907} C_VEL
LIN {X 0,Y 594.874,Z 433.901,A -85,B 0,C 180,E1 -1155.57,E2 -1155.57} C_VEL
LIN {X 0,Y 594.818,Z 448.155,A -85,B 0,C 180,E1 -1155.889,E2 -1155.889} C_VEL
LIN {X 0,Y 594.729,Z 461.721,A -85,B 0,C 180,E1 -1156.329,E2 -1156.329} C_VEL
LIN {X 0,Y 594.653,Z 475.642,A -85,B 0,C 180,E1 -1156.937,E2 -1156.937} C_VEL
LIN {X 0,Y 594.581,Z 488.1,A -85,B 0,C 180,E1 -1157.629,E2 -1157.629} C_VEL
LIN {X 0,Y 594.524,Z 500.562,A -85,B 0,C 180,E1 -1158.488,E2 -1158.488} C_VEL
LIN {X 0,Y 594.449,Z 511.839,A -85,B 0,C 180,E1 -1159.441,E2 -1159.441} C_VEL
LIN {X 0,Y 594.368,Z 521.852,A -85,B 0,C 180,E1 -1160.472,E2 -1160.472} C_VEL
LIN {X 0,Y 594.324,Z 530.172,A -85,B 0,C 180,E1 -1161.5,E2 -1161.5} C_VEL
LIN {X 0,Y 594.303,Z 538.126,A -85,B 0,C 180,E1 -1162.697,E2 -1162.697} C_VEL
LIN {X 0,Y 594.281,Z 544.528,A -85,B 0,C 180,E1 -1163.89,E2 -1163.89} C_VEL
LIN {X 0,Y 594.237,Z 550.199,A -85,B 0,C 180,E1 -1165.251,E2 -1165.251} C_VEL
LIN {X 0,Y 594.259,Z 554.315,A -85,B 0,C 180,E1 -1166.61,E2 -1166.61} C_VEL
LIN {X 0,Y 594.241,Z 557,A -85,B 0,C 180,E1 -1167.967,E2 -1167.967} C_VEL
LIN {X 0,Y 594.237,Z 558.332,A -85,B 0,C 180,E1 -1169.322,E2 -1169.322} C_VEL
LIN {X 0,Y 594.237,Z 558.332,A -85,B 0,C 180,E1 -1170.678,E2 -1170.678} C_VEL
LIN {X 0,Y 594.242,Z 557,A -85,B 0,C 180,E1 -1172.033,E2 -1172.033} C_VEL
LIN {X 0,Y 594.259,Z 554.316,A -85,B 0,C 180,E1 -1173.39,E2 -1173.39} C_VEL
LIN {X 0,Y 594.237,Z 550.199,A -85,B 0,C 180,E1 -1174.749,E2 -1174.749} C_VEL
LIN {X 0,Y 594.281,Z 544.527,A -85,B 0,C 180,E1 -1176.11,E2 -1176.11} C_VEL
LIN {X 0,Y 594.303,Z 538.126,A -85,B 0,C 180,E1 -1177.303,E2 -1177.303} C_VEL
LIN {X 0,Y 594.324,Z 530.171,A -85,B 0,C 180,E1 -1178.5,E2 -1178.5} C_VEL
LIN {X 0,Y 594.367,Z 521.851,A -85,B 0,C 180,E1 -1179.529,E2 -1179.529} C_VEL
LIN {X 0,Y 594.449,Z 511.838,A -85,B 0,C 180,E1 -1180.559,E2 -1180.559} C_VEL
LIN {X 0,Y 594.523,Z 500.564,A -85,B 0,C 180,E1 -1181.512,E2 -1181.512} C_VEL
LIN {X 0,Y 594.58,Z 488.099,A -85,B 0,C 180,E1 -1182.371,E2 -1182.371} C_VEL
LIN {X 0,Y 594.653,Z 475.641,A -85,B 0,C 180,E1 -1183.063,E2 -1183.063} C_VEL
LIN {X 0,Y 594.743,Z 461.716,A -85,B 0,C 180,E1 -1183.67,E2 -1183.67} C_VEL
LIN {X 0,Y 594.819,Z 448.135,A -85,B 0,C 180,E1 -1184.112,E2 -1184.112} C_VEL
LIN {X 0,Y 594.873,Z 433.895,A -85,B 0,C 180,E1 -1184.43,E2 -1184.43} C_VEL
LIN {X 0,Y 594.929,Z 296.73,A -85,B 0,C 180,E1 -1186.131,E2 -1186.131} C_VEL
LIN {X 0,Y 594.617,Z 294.66,A -85,B 0,C 180,E1 -1186.192,E2 -1186.192} C_VEL
LIN {X 0,Y 594.695,Z 269.257,A -85,B 0,C 180,E1 -1189.016,E2 -1189.016} C_VEL
LIN {X 0,Y 594.888,Z 245.882,A -85,B 0,C 180,E1 -1191.665,E2 -1191.665} C_VEL
LIN {X 0,Y 594.761,Z 235.841,A -85,B 0,C 180,E1 -1192.826,E2 -1192.826} C_VEL
LIN {X 0,Y 594.385,Z 234.132,A -85,B 0,C 180,E1 -1193.081,E2 -1193.081} C_VEL
LIN {X 0,Y 594.377,Z 234.069,A -85,B 0,C 180,E1 -1195.193,E2 -1195.193} C_VEL
LIN {X 0,Y 594.385,Z 234.066,A -85,B 0,C 180,E1 -1197.526,E2 -1197.526} C_VEL
LIN {X 0,Y 594.384,Z 234.073,A -85,B 0,C 180,E1 -1200.328,E2 -1200.328} C_VEL
LIN {X 0,Y 594.379,Z 234.069,A -85,B 0,C 180,E1 -1202.95,E2 -1202.95} C_VEL
LIN {X 0,Y 594.348,Z 234.069,A -85,B 0,C 180,E1 -1205.408,E2 -1205.408} C_VEL
LIN {X 0,Y 594.383,Z 234.068,A -85,B 0,C 180,E1 -1207.94,E2 -1207.94} C_VEL
LIN {X 0,Y 594.377,Z 234.069,A -85,B 0,C 180,E1 -1210.822,E2 -1210.822} C_VEL
LIN {X 0,Y 594.379,Z 234.069,A -85,B 0,C 180,E1 -1213.841,E2 -1213.841} C_VEL
LIN {X 0,Y 594.362,Z 234.071,A -85,B 0,C 180,E1 -1216.7,E2 -1216.7} C_VEL
LIN {X 0,Y 594.366,Z 234.067,A -85,B 0,C 180,E1 -1219.433,E2 -1219.433} C_VEL
LIN {X 0,Y 594.385,Z 234.071,A -85,B 0,C 180,E1 -1222.391,E2 -1222.391} C_VEL
LIN {X 0,Y 594.38,Z 234.067,A -85,B 0,C 180,E1 -1224.671,E2 -1224.671} C_VEL
LIN {X 0,Y 594.372,Z 234.067,A -85,B 0,C 180,E1 -1227.088,E2 -1227.088} C_VEL
LIN {X 0,Y 594.395,Z 234.067,A -85,B 0,C 180,E1 -1229.669,E2 -1229.669} C_VEL
LIN {X 0,Y 594.385,Z 234.067,A -85,B 0,C 180,E1 -1232.54,E2 -1232.54} C_VEL
LIN {X 0,Y 594.392,Z 234.068,A -85,B 0,C 180,E1 -1235.564,E2 -1235.564} C_VEL
LIN {X 0,Y 594.362,Z 234.069,A -85,B 0,C 180,E1 -1238.497,E2 -1238.497} C_VEL
LIN {X 0,Y 594.378,Z 234.069,A -85,B 0,C 180,E1 -1241.383,E2 -1241.383} C_VEL
LIN {X 0,Y 594.366,Z 234.071,A -85,B 0,C 180,E1 -1244.219,E2 -1244.219} C_VEL
LIN {X 0,Y 594.367,Z 234.068,A -85,B 0,C 180,E1 -1247.017,E2 -1247.017} C_VEL
LIN {X 0,Y 594.387,Z 234.074,A -85,B 0,C 180,E1 -1249.784,E2 -1249.784} C_VEL
LIN {X 0,Y 594.396,Z 234.063,A -85,B 0,C 180,E1 -1252.527,E2 -1252.527} C_VEL
LIN {X 0,Y 594.39,Z 234.069,A -85,B 0,C 180,E1 -1255.253,E2 -1255.253} C_VEL
LIN {X 0,Y 594.39,Z 234.068,A -85,B 0,C 180,E1 -1257.967,E2 -1257.967} C_VEL
LIN {X 0,Y 594.417,Z 234.061,A -85,B 0,C 180,E1 -1260.678,E2 -1260.678} C_VEL
LIN {X 0,Y 594.379,Z 234.074,A -85,B 0,C 180,E1 -1263.39,E2 -1263.39} C_VEL
LIN {X 0,Y 594.363,Z 234.068,A -85,B 0,C 180,E1 -1266.109,E2 -1266.109} C_VEL
LIN {X 0,Y 594.395,Z 234.066,A -85,B 0,C 180,E1 -1268.842,E2 -1268.842} C_VEL
LIN {X 0,Y 594.388,Z 234.07,A -85,B 0,C 180,E1 -1271.596,E2 -1271.596} C_VEL
LIN {X 0,Y 594.383,Z 234.065,A -85,B 0,C 180,E1 -1274.378,E2 -1274.378} C_VEL
LIN {X 0,Y 594.357,Z 234.072,A -85,B 0,C 180,E1 -1275.333,E2 -1275.333} C_VEL
LIN {X 0,Y 593.687,Z 234.154,A -85,B 0,C 180,E1 -1275.899,E2 -1275.899} C_VEL
LIN {X 0,Y 590.834,Z 234.51,A -85,B 0,C 180,E1 -1276.817,E2 -1276.817} C_VEL
LIN {X 0,Y 588.428,Z 234.812,A -85,B 0,C 180,E1 -1277.556,E2 -1277.556} C_VEL
LIN {X 0,Y 587.4,Z 234.936,A -85,B 0,C 180,E1 -1278.126,E2 -1278.126} C_VEL
LIN {X 0,Y 587.319,Z 234.945,A -85,B 0,C 180,E1 -1278.319,E2 -1278.319} C_VEL
LIN {X 0,Y 587.324,Z 234.951,A -85,B 0,C 180,E1 -1281.038,E2 -1281.038} C_VEL
LIN {X 0,Y 587.318,Z 234.954,A -85,B 0,C 180,E1 -1283.259,E2 -1283.259} C_VEL
LIN {X 0,Y 587.331,Z 234.948,A -85,B 0,C 180,E1 -1285.517,E2 -1285.517} C_VEL
LIN {X 0,Y 587.344,Z 234.942,A -85,B 0,C 180,E1 -1287.818,E2 -1287.818} C_VEL
LIN {X 0,Y 587.339,Z 234.944,A -85,B 0,C 180,E1 -1290.512,E2 -1290.512} C_VEL
LIN {X 0,Y 587.335,Z 234.951,A -85,B 0,C 180,E1 -1293.113,E2 -1293.113} C_VEL
LIN {X 0,Y 587.354,Z 234.94,A -85,B 0,C 180,E1 -1295.896,E2 -1295.896} C_VEL
LIN {X 0,Y 587.332,Z 234.947,A -85,B 0,C 180,E1 -1298.48,E2 -1298.48} C_VEL
LIN {X 0,Y 587.334,Z 234.949,A -85,B 0,C 180,E1 -1301.158,E2 -1301.158} C_VEL
LIN {X 0,Y 587.325,Z 234.945,A -85,B 0,C 180,E1 -1304.114,E2 -1304.114} C_VEL
LIN {X 0,Y 587.323,Z 234.951,A -85,B 0,C 180,E1 -1306.995,E2 -1306.995} C_VEL
LIN {X 0,Y 587.312,Z 234.946,A -85,B 0,C 180,E1 -1309.746,E2 -1309.746} C_VEL
LIN {X 0,Y 587.345,Z 234.944,A -85,B 0,C 180,E1 -1312.393,E2 -1312.393} C_VEL
LIN {X 0,Y 587.342,Z 234.941,A -85,B 0,C 180,E1 -1315.654,E2 -1315.654} C_VEL
LIN {X 0,Y 587.344,Z 234.947,A -85,B 0,C 180,E1 -1318.232,E2 -1318.232} C_VEL
LIN {X 0,Y 587.351,Z 234.946,A -85,B 0,C 180,E1 -1320.867,E2 -1320.867} C_VEL
LIN {X 0,Y 587.363,Z 235.009,A -85,B 0,C 180,E1 -1323.819,E2 -1323.819} C_VEL
LIN {X 0,Y 587.47,Z 235.696,A -85,B 0,C 180,E1 -1324.005,E2 -1324.005} C_VEL
LIN {X 0,Y 587.991,Z 239.256,A -85,B 0,C 180,E1 -1324.514,E2 -1324.514} C_VEL
LIN {X 0,Y 587.817,Z 259.784,A -85,B 0,C 180,E1 -1327.262,E2 -1327.262} C_VEL
LIN {X 0,Y 587.659,Z 279.755,A -85,B 0,C 180,E1 -1329.89,E2 -1329.89} C_VEL
LIN {X 0,Y 587.53,Z 301.932,A -85,B 0,C 180,E1 -1332.766,E2 -1332.766} C_VEL
LIN {X 0,Y 587.437,Z 315.789,A -85,B 0,C 180,E1 -1334.518,E2 -1334.518} C_VEL
LIN {X 0,Y 587.867,Z 319.251,A -85,B 0,C 180,E1 -1334.596,E2 -1334.596} C_VEL
LIN {X 0,Y 587.743,Z 424.643,A -85,B 0,C 180,E1 -1335.904,E2 -1335.904} C_VEL
LIN {X 0,Y 587.683,Z 437.748,A -85,B 0,C 180,E1 -1336.206,E2 -1336.206} C_VEL
LIN {X 0,Y 587.641,Z 450.526,A -85,B 0,C 180,E1 -1336.646,E2 -1336.646} C_VEL
LIN {X 0,Y 587.506,Z 462.665,A -85,B 0,C 180,E1 -1337.215,E2 -1337.215} C_VEL
LIN {X 0,Y 587.458,Z 474.203,A -85,B 0,C 180,E1 -1337.915,E2 -1337.915} C_VEL
LIN {X 0,Y 587.378,Z 485.045,A -85,B 0,C 180,E1 -1338.741,E2 -1338.741} C_VEL
LIN {X 0,Y 587.337,Z 494.701,A -85,B 0,C 180,E1 -1339.66,E2 -1339.66} C_VEL
LIN {X 0,Y 587.272,Z 503.576,A -85,B 0,C 180,E1 -1340.703,E2 -1340.703} C_VEL
LIN {X 0,Y 587.232,Z 510.672,A -85,B 0,C 180,E1 -1341.743,E2 -1341.743} C_VEL
LIN {X 0,Y 587.215,Z 516.33,A -85,B 0,C 180,E1 -1342.781,E2 -1342.781} C_VEL
LIN {X 0,Y 587.169,Z 520.778,A -85,B 0,C 180,E1 -1343.816,E2 -1343.816} C_VEL
LIN {X 0,Y 587.191,Z 523.124,A -85,B 0,C 180,E1 -1344.506,E2 -1344.506} C_VEL
LIN {X 0,Y 587.131,Z 525.037,A -85,B 0,C 180,E1 -1345.194,E2 -1345.194} C_VEL
LIN {X 0,Y 587.171,Z 526.526,A -85,B 0,C 180,E1 -1345.882,E2 -1345.882} C_VEL
LIN {X 0,Y 587.182,Z 527.567,A -85,B 0,C 180,E1 -1346.569,E2 -1346.569} C_VEL
LIN {X 0,Y 587.14,Z 528.483,A -85,B 0,C 180,E1 -1347.942,E2 -1347.942} C_VEL
LIN {X 0,Y 587.147,Z 528.354,A -85,B 0,C 180,E1 -1348.628,E2 -1348.628} C_VEL
LIN {X 0,Y 587.139,Z 526.869,A -85,B 0,C 180,E1 -1350,E2 -1350} C_VEL
LIN {X 0,Y 587.14,Z 525.539,A -85,B 0,C 180,E1 -1350.686,E2 -1350.686} C_VEL
LIN {X 0,Y 587.18,Z 522.722,A -85,B 0,C 180,E1 -1351.715,E2 -1351.715} C_VEL
LIN {X 0,Y 587.153,Z 518.892,A -85,B 0,C 180,E1 -1352.744,E2 -1352.744} C_VEL
LIN {X 0,Y 587.214,Z 513.944,A -85,B 0,C 180,E1 -1353.774,E2 -1353.774} C_VEL
LIN {X 0,Y 587.28,Z 507.731,A -85,B 0,C 180,E1 -1354.805,E2 -1354.805} C_VEL
LIN {X 0,Y 587.267,Z 499.985,A -85,B 0,C 180,E1 -1355.838,E2 -1355.838} C_VEL
LIN {X 0,Y 587.336,Z 490.306,A -85,B 0,C 180,E1 -1356.872,E2 -1356.872} C_VEL
LIN {X 0,Y 587.414,Z 480.283,A -85,B 0,C 180,E1 -1357.735,E2 -1357.735} C_VEL
LIN {X 0,Y 587.522,Z 468.964,A -85,B 0,C 180,E1 -1358.513,E2 -1358.513} C_VEL
LIN {X 0,Y 587.572,Z 457.858,A -85,B 0,C 180,E1 -1359.119,E2 -1359.119} C_VEL
LIN {X 0,Y 587.681,Z 445.448,A -85,B 0,C 180,E1 -1359.638,E2 -1359.638} C_VEL
LIN {X 0,Y 587.722,Z 432.211,A -85,B 0,C 180,E1 -1360.028,E2 -1360.028} C_VEL
LIN {X 0,Y 587.78,Z 419.271,A -85,B 0,C 180,E1 -1360.267,E2 -1360.267} C_VEL
LIN {X 0,Y 587.758,Z 318.074,A -85,B 0,C 180,E1 -1361.511,E2 -1361.511} C_VEL
LIN {X 0,Y 587.475,Z 315.768,A -85,B 0,C 180,E1 -1361.573,E2 -1361.573} C_VEL
LIN {X 0,Y 587.559,Z 294.128,A -85,B 0,C 180,E1 -1364.332,E2 -1364.332} C_VEL
LIN {X 0,Y 587.726,Z 270.643,A -85,B 0,C 180,E1 -1367.394,E2 -1367.394} C_VEL
LIN {X 0,Y 587.856,Z 250.222,A -85,B 0,C 180,E1 -1370.103,E2 -1370.103} C_VEL
LIN {X 0,Y 587.942,Z 237.987,A -85,B 0,C 180,E1 -1371.75,E2 -1371.75} C_VEL
LIN {X 0,Y 587.36,Z 235.073,A -85,B 0,C 180,E1 -1372.211,E2 -1372.211} C_VEL
LIN {X 0,Y 587.354,Z 234.941,A -85,B 0,C 180,E1 -1374.758,E2 -1374.758} C_VEL
LIN {X 0,Y 587.331,Z 234.945,A -85,B 0,C 180,E1 -1377.046,E2 -1377.046} C_VEL
LIN {X 0,Y 587.349,Z 234.95,A -85,B 0,C 180,E1 -1379.379,E2 -1379.379} C_VEL
LIN {X 0,Y 587.347,Z 234.946,A -85,B 0,C 180,E1 -1381.835,E2 -1381.835} C_VEL
LIN {X 0,Y 587.348,Z 234.94,A -85,B 0,C 180,E1 -1384.347,E2 -1384.347} C_VEL
LIN {X 0,Y 587.344,Z 234.948,A -85,B 0,C 180,E1 -1387.607,E2 -1387.607} C_VEL
LIN {X 0,Y 587.311,Z 234.946,A -85,B 0,C 180,E1 -1390.254,E2 -1390.254} C_VEL
LIN {X 0,Y 587.323,Z 234.951,A -85,B 0,C 180,E1 -1393.005,E2 -1393.005} C_VEL
LIN {X 0,Y 587.325,Z 234.945,A -85,B 0,C 180,E1 -1395.886,E2 -1395.886} C_VEL
LIN {X 0,Y 587.334,Z 234.95,A -85,B 0,C 180,E1 -1398.924,E2 -1398.924} C_VEL
LIN {X 0,Y 587.331,Z 234.947,A -85,B 0,C 180,E1 -1401.52,E2 -1401.52} C_VEL
LIN {X 0,Y 587.348,Z 234.943,A -85,B 0,C 180,E1 -1404.454,E2 -1404.454} C_VEL
LIN {X 0,Y 587.335,Z 234.949,A -85,B 0,C 180,E1 -1406.887,E2 -1406.887} C_VEL
LIN {X 0,Y 587.347,Z 234.944,A -85,B 0,C 180,E1 -1409.487,E2 -1409.487} C_VEL
LIN {X 0,Y 587.346,Z 234.943,A -85,B 0,C 180,E1 -1412.306,E2 -1412.306} C_VEL
LIN {X 0,Y 587.33,Z 234.948,A -85,B 0,C 180,E1 -1414.483,E2 -1414.483} C_VEL
LIN {X 0,Y 587.313,Z 234.952,A -85,B 0,C 180,E1 -1417.131,E2 -1417.131} C_VEL
LIN {X 0,Y 587.326,Z 234.944,A -85,B 0,C 180,E1 -1419.695,E2 -1419.695} C_VEL
LIN {X 0,Y 587.354,Z 234.948,A -85,B 0,C 180,E1 -1422.594,E2 -1422.594} C_VEL
LIN {X 0,Y 587.358,Z 234.94,A -85,B 0,C 180,E1 -1425.739,E2 -1425.739} C_VEL
LIN {X 0,Y 587.34,Z 234.948,A -85,B 0,C 180,E1 -1428.866,E2 -1428.866} C_VEL
LIN {X 0,Y 587.363,Z 234.94,A -85,B 0,C 180,E1 -1431.744,E2 -1431.744} C_VEL
LIN {X 0,Y 587.354,Z 234.95,A -85,B 0,C 180,E1 -1434.507,E2 -1434.507} C_VEL
LIN {X 0,Y 587.373,Z 234.939,A -85,B 0,C 180,E1 -1437.257,E2 -1437.257} C_VEL
LIN {X 0,Y 587.375,Z 234.941,A -85,B 0,C 180,E1 -1440,E2 -1440} C_VEL
LIN {X 0,Y 587.371,Z 234.944,A -85,B 0,C 180,E1 -1442.743,E2 -1442.743} C_VEL
LIN {X 0,Y 587.355,Z 234.94,A -85,B 0,C 180,E1 -1445.493,E2 -1445.493} C_VEL
LIN {X 0,Y 587.364,Z 234.948,A -85,B 0,C 180,E1 -1448.255,E2 -1448.255} C_VEL
LIN {X 0,Y 587.339,Z 234.942,A -85,B 0,C 180,E1 -1451.134,E2 -1451.134} C_VEL
LIN {X 0,Y 587.355,Z 234.945,A -85,B 0,C 180,E1 -1453.846,E2 -1453.846} C_VEL
LIN {X 0,Y 587.355,Z 234.942,A -85,B 0,C 180,E1 -1456.819,E2 -1456.819} C_VEL
LIN {X 0,Y 587.339,Z 234.945,A -85,B 0,C 180,E1 -1459.575,E2 -1459.575} C_VEL
LIN {X 0,Y 587.334,Z 234.947,A -85,B 0,C 180,E1 -1462.514,E2 -1462.514} C_VEL
LIN {X 0,Y 587.345,Z 234.942,A -85,B 0,C 180,E1 -1464.759,E2 -1464.759} C_VEL
LIN {X 0,Y 587.333,Z 234.943,A -85,B 0,C 180,E1 -1467.046,E2 -1467.046} C_VEL
LIN {X 0,Y 587.345,Z 234.943,A -85,B 0,C 180,E1 -1469.38,E2 -1469.38} C_VEL
LIN {X 0,Y 587.348,Z 234.948,A -85,B 0,C 180,E1 -1471.838,E2 -1471.838} C_VEL
LIN {X 0,Y 587.351,Z 234.945,A -85,B 0,C 180,E1 -1474.35,E2 -1474.35} C_VEL
LIN {X 0,Y 587.348,Z 234.94,A -85,B 0,C 180,E1 -1476.747,E2 -1476.747} C_VEL
LIN {X 0,Y 587.342,Z 234.945,A -85,B 0,C 180,E1 -1479.36,E2 -1479.36} C_VEL
LIN {X 0,Y 587.33,Z 234.948,A -85,B 0,C 180,E1 -1482.108,E2 -1482.108} C_VEL
LIN {X 0,Y 587.311,Z 234.948,A -85,B 0,C 180,E1 -1485.089,E2 -1485.089} C_VEL
LIN {X 0,Y 587.349,Z 234.944,A -85,B 0,C 180,E1 -1487.928,E2 -1487.928} C_VEL
LIN {X 0,Y 587.321,Z 234.947,A -85,B 0,C 180,E1 -1491.06,E2 -1491.06} C_VEL
LIN {X 0,Y 587.344,Z 234.947,A -85,B 0,C 180,E1 -1493.293,E2 -1493.293} C_VEL
LIN {X 0,Y 587.36,Z 234.947,A -85,B 0,C 180,E1 -1495.781,E2 -1495.781} C_VEL
LIN {X 0,Y 587.346,Z 234.941,A -85,B 0,C 180,E1 -1498.232,E2 -1498.232} C_VEL
LIN {X 0,Y 587.349,Z 234.944,A -85,B 0,C 180,E1 -1500.867,E2 -1500.867} C_VEL
LIN {X 0,Y 587.36,Z 234.945,A -85,B 0,C 180,E1 -1503.819,E2 -1503.819} C_VEL
LIN {X 0,Y 587.363,Z 235.039,A -85,B 0,C 180,E1 -1506.743,E2 -1506.743} C_VEL
LIN {X 0,Y 588.088,Z 239.671,A -85,B 0,C 180,E1 -1507.348,E2 -1507.348} C_VEL
LIN {X 0,Y 587.876,Z 264.948,A -85,B 0,C 180,E1 -1510.262,E2 -1510.262} C_VEL
LIN {X 0,Y 587.624,Z 289.988,A -85,B 0,C 180,E1 -1513.098,E2 -1513.098} C_VEL
LIN {X 0,Y 587.68,Z 295.038,A -85,B 0,C 180,E1 -1513.634,E2 -1513.634} C_VEL
LIN {X 0,Y 588.203,Z 299.642,A -85,B 0,C 180,E1 -1513.716,E2 -1513.716} C_VEL
LIN {X 0,Y 588.014,Z 433.9,A -85,B 0,C 180,E1 -1515.398,E2 -1515.398} C_VEL
LIN {X 0,Y 587.942,Z 447.502,A -85,B 0,C 180,E1 -1515.701,E2 -1515.701} C_VEL
LIN {X 0,Y 587.817,Z 461.72,A -85,B 0,C 180,E1 -1516.166,E2 -1516.166} C_VEL
LIN {X 0,Y 587.731,Z 475.645,A -85,B 0,C 180,E1 -1516.78,E2 -1516.78} C_VEL
LIN {X 0,Y 587.605,Z 488.102,A -85,B 0,C 180,E1 -1517.48,E2 -1517.48} C_VEL
LIN {X 0,Y 587.513,Z 500.642,A -85,B 0,C 180,E1 -1518.354,E2 -1518.354} C_VEL
LIN {X 0,Y 587.444,Z 511.838,A -85,B 0,C 180,E1 -1519.314,E2 -1519.314} C_VEL
LIN {X 0,Y 587.319,Z 521.852,A -85,B 0,C 180,E1 -1520.356,E2 -1520.356} C_VEL
LIN {X 0,Y 587.277,Z 530.172,A -85,B 0,C 180,E1 -1521.397,E2 -1521.397} C_VEL
LIN {X 0,Y 587.244,Z 538.127,A -85,B 0,C 180,E1 -1522.608,E2 -1522.608} C_VEL
LIN {X 0,Y 587.204,Z 544.528,A -85,B 0,C 180,E1 -1523.816,E2 -1523.816} C_VEL
LIN {X 0,Y 587.16,Z 548.962,A -85,B 0,C 180,E1 -1524.85,E2 -1524.85} C_VEL
LIN {X 0,Y 587.179,Z 552.443,A -85,B 0,C 180,E1 -1525.882,E2 -1525.882} C_VEL
LIN {X 0,Y 587.13,Z 555.832,A -85,B 0,C 180,E1 -1527.256,E2 -1527.256} C_VEL
LIN {X 0,Y 587.142,Z 557.832,A -85,B 0,C 180,E1 -1528.628,E2 -1528.628} C_VEL
LIN {X 0,Y 587.135,Z 558.5,A -85,B 0,C 180,E1 -1530,E2 -1530} C_VEL
LIN {X 0,Y 587.142,Z 557.832,A -85,B 0,C 180,E1 -1531.372,E2 -1531.372} C_VEL
LIN {X 0,Y 587.13,Z 555.833,A -85,B 0,C 180,E1 -1532.744,E2 -1532.744} C_VEL
LIN {X 0,Y 587.179,Z 552.444,A -85,B 0,C 180,E1 -1534.118,E2 -1534.118} C_VEL
LIN {X 0,Y 587.2,Z 547.568,A -85,B 0,C 180,E1 -1535.494,E2 -1535.494} C_VEL
LIN {X 0,Y 587.209,Z 541.053,A -85,B 0,C 180,E1 -1536.874,E2 -1536.874} C_VEL
LIN {X 0,Y 587.268,Z 533.8,A -85,B 0,C 180,E1 -1538.083,E2 -1538.083} C_VEL
LIN {X 0,Y 587.321,Z 524.824,A -85,B 0,C 180,E1 -1539.296,E2 -1539.296} C_VEL
LIN {X 0,Y 587.372,Z 515.393,A -85,B 0,C 180,E1 -1540.339,E2 -1540.339} C_VEL
LIN {X 0,Y 587.475,Z 505.028,A -85,B 0,C 180,E1 -1541.29,E2 -1541.29} C_VEL
LIN {X 0,Y 587.577,Z 493.433,A -85,B 0,C 180,E1 -1542.17,E2 -1542.17} C_VEL
LIN {X 0,Y 587.67,Z 480.651,A -85,B 0,C 180,E1 -1542.958,E2 -1542.958} C_VEL
LIN {X 0,Y 587.799,Z 468.163,A -85,B 0,C 180,E1 -1543.571,E2 -1543.571} C_VEL
LIN {X 0,Y 587.917,Z 454.611,A -85,B 0,C 180,E1 -1544.085,E2 -1544.085} C_VEL
LIN {X 0,Y 587.989,Z 440.693,A -85,B 0,C 180,E1 -1544.467,E2 -1544.467} C_VEL
LIN {X 0,Y 588.017,Z 426.618,A -85,B 0,C 180,E1 -1544.713,E2 -1544.713} C_VEL
LIN {X 0,Y 588.131,Z 297.847,A -85,B 0,C 180,E1 -1546.309,E2 -1546.309} C_VEL
LIN {X 0,Y 587.655,Z 294.669,A -85,B 0,C 180,E1 -1546.389,E2 -1546.389} C_VEL
LIN {X 0,Y 587.812,Z 268.842,A -85,B 0,C 180,E1 -1549.295,E2 -1549.295} C_VEL
LIN {X 0,Y 588.076,Z 242.705,A -85,B 0,C 180,E1 -1552.299,E2 -1552.299} C_VEL
LIN {X 0,Y 587.782,Z 237.013,A -85,B 0,C 180,E1 -1552.975,E2 -1552.975} C_VEL
LIN {X 0,Y 587.363,Z 235.038,A -85,B 0,C 180,E1 -1553.257,E2 -1553.257} C_VEL
LIN {X 0,Y 587.36,Z 234.945,A -85,B 0,C 180,E1 -1556.181,E2 -1556.181} C_VEL
LIN {X 0,Y 587.349,Z 234.943,A -85,B 0,C 180,E1 -1559.133,E2 -1559.133} C_VEL
LIN {X 0,Y 587.345,Z 234.942,A -85,B 0,C 180,E1 -1561.836,E2 -1561.836} C_VEL
LIN {X 0,Y 587.347,Z 234.951,A -85,B 0,C 180,E1 -1564.347,E2 -1564.347} C_VEL
LIN {X 0,Y 587.342,Z 234.941,A -85,B 0,C 180,E1 -1567.607,E2 -1567.607} C_VEL
LIN {X 0,Y 587.311,Z 234.955,A -85,B 0,C 180,E1 -1570.254,E2 -1570.254} C_VEL
LIN {X 0,Y 587.321,Z 234.946,A -85,B 0,C 180,E1 -1573.005,E2 -1573.005} C_VEL
LIN {X 0,Y 587.322,Z 234.949,A -85,B 0,C 180,E1 -1575.886,E2 -1575.886} C_VEL
LIN {X 0,Y 587.332,Z 234.944,A -85,B 0,C 180,E1 -1578.843,E2 -1578.843} C_VEL
LIN {X 0,Y 587.329,Z 234.946,A -85,B 0,C 180,E1 -1581.521,E2 -1581.521} C_VEL
LIN {X 0,Y 587.347,Z 234.946,A -85,B 0,C 180,E1 -1584.454,E2 -1584.454} C_VEL
LIN {X 0,Y 587.333,Z 234.944,A -85,B 0,C 180,E1 -1586.888,E2 -1586.888} C_VEL
LIN {X 0,Y 587.345,Z 234.943,A -85,B 0,C 180,E1 -1589.487,E2 -1589.487} C_VEL
LIN {X 0,Y 587.345,Z 234.947,A -85,B 0,C 180,E1 -1592.307,E2 -1592.307} C_VEL
LIN {X 0,Y 587.345,Z 234.943,A -85,B 0,C 180,E1 -1595.241,E2 -1595.241} C_VEL
LIN {X 0,Y 587.318,Z 234.95,A -85,B 0,C 180,E1 -1598.226,E2 -1598.226} C_VEL
LIN {X 0,Y 587.342,Z 234.943,A -85,B 0,C 180,E1 -1601.151,E2 -1601.151} C_VEL
LIN {X 0,Y 587.346,Z 234.944,A -85,B 0,C 180,E1 -1603.311,E2 -1603.311} C_VEL
LIN {X 0,Y 587.356,Z 234.944,A -85,B 0,C 180,E1 -1606.154,E2 -1606.154} C_VEL
LIN {X 0,Y 587.335,Z 234.943,A -85,B 0,C 180,E1 -1608.962,E2 -1608.962} C_VEL
LIN {X 0,Y 587.364,Z 234.948,A -85,B 0,C 180,E1 -1611.745,E2 -1611.745} C_VEL
LIN {X 0,Y 587.355,Z 234.941,A -85,B 0,C 180,E1 -1614.507,E2 -1614.507} C_VEL
LIN {X 0,Y 587.371,Z 234.943,A -85,B 0,C 180,E1 -1617.257,E2 -1617.257} C_VEL
LIN {X 0,Y 587.376,Z 234.941,A -85,B 0,C 180,E1 -1620,E2 -1620} C_VEL
LIN {X 0,Y 587.373,Z 234.938,A -85,B 0,C 180,E1 -1622.743,E2 -1622.743} C_VEL
LIN {X 0,Y 587.354,Z 234.95,A -85,B 0,C 180,E1 -1625.493,E2 -1625.493} C_VEL
LIN {X 0,Y 587.364,Z 234.94,A -85,B 0,C 180,E1 -1628.256,E2 -1628.256} C_VEL
LIN {X 0,Y 587.341,Z 234.949,A -85,B 0,C 180,E1 -1631.134,E2 -1631.134} C_VEL
LIN {X 0,Y 587.359,Z 234.94,A -85,B 0,C 180,E1 -1634.261,E2 -1634.261} C_VEL
LIN {X 0,Y 587.354,Z 234.949,A -85,B 0,C 180,E1 -1637.406,E2 -1637.406} C_VEL
LIN {X 0,Y 587.319,Z 234.945,A -85,B 0,C 180,E1 -1638.319,E2 -1638.319} C_VEL
LIN {X 0,Y 586.665,Z 235.032,A -85,B 0,C 180,E1 -1638.891,E2 -1638.891} C_VEL
LIN {X 0,Y 583.832,Z 235.392,A -85,B 0,C 180,E1 -1639.819,E2 -1639.819} C_VEL
LIN {X 0,Y 581.423,Z 235.695,A -85,B 0,C 180,E1 -1640.566,E2 -1640.566} C_VEL
LIN {X 0,Y 580.371,Z 235.822,A -85,B 0,C 180,E1 -1641.142,E2 -1641.142} C_VEL
LIN {X 0,Y 580.277,Z 235.83,A -85,B 0,C 180,E1 -1641.338,E2 -1641.338} C_VEL
LIN {X 0,Y 580.297,Z 235.82,A -85,B 0,C 180,E1 -1644.317,E2 -1644.317} C_VEL
LIN {X 0,Y 580.274,Z 235.826,A -85,B 0,C 180,E1 -1646.624,E2 -1646.624} C_VEL
LIN {X 0,Y 580.298,Z 235.825,A -85,B 0,C 180,E1 -1649.311,E2 -1649.311} C_VEL
LIN {X 0,Y 580.298,Z 235.82,A -85,B 0,C 180,E1 -1652.201,E2 -1652.201} C_VEL
LIN {X 0,Y 580.297,Z 235.825,A -85,B 0,C 180,E1 -1654.696,E2 -1654.696} C_VEL
LIN {X 0,Y 580.298,Z 235.825,A -85,B 0,C 180,E1 -1657.269,E2 -1657.269} C_VEL
LIN {X 0,Y 580.295,Z 235.82,A -85,B 0,C 180,E1 -1660.272,E2 -1660.272} C_VEL
LIN {X 0,Y 580.276,Z 235.831,A -85,B 0,C 180,E1 -1662.707,E2 -1662.707} C_VEL
LIN {X 0,Y 580.274,Z 235.824,A -85,B 0,C 180,E1 -1665.609,E2 -1665.609} C_VEL
LIN {X 0,Y 580.314,Z 235.819,A -85,B 0,C 180,E1 -1668.235,E2 -1668.235} C_VEL
LIN {X 0,Y 580.278,Z 235.824,A -85,B 0,C 180,E1 -1670.966,E2 -1670.966} C_VEL
LIN {X 0,Y 580.268,Z 235.824,A -85,B 0,C 180,E1 -1673.597,E2 -1673.597} C_VEL
LIN {X 0,Y 580.301,Z 235.821,A -85,B 0,C 180,E1 -1676.145,E2 -1676.145} C_VEL
LIN {X 0,Y 580.277,Z 235.83,A -85,B 0,C 180,E1 -1678.615,E2 -1678.615} C_VEL
LIN {X 0,Y 580.294,Z 235.823,A -85,B 0,C 180,E1 -1681.025,E2 -1681.025} C_VEL
LIN {X 0,Y 580.322,Z 235.925,A -85,B 0,C 180,E1 -1683.688,E2 -1683.688} C_VEL
LIN {X 0,Y 581.088,Z 240.426,A -85,B 0,C 180,E1 -1684.382,E2 -1684.382} C_VEL
LIN {X 0,Y 580.897,Z 259.484,A -85,B 0,C 180,E1 -1686.963,E2 -1686.963} C_VEL
LIN {X 0,Y 580.712,Z 279.557,A -85,B 0,C 180,E1 -1689.639,E2 -1689.639} C_VEL
LIN {X 0,Y 580.536,Z 301.982,A -85,B 0,C 180,E1 -1692.583,E2 -1692.583} C_VEL
LIN {X 0,Y 580.437,Z 315.769,A -85,B 0,C 180,E1 -1694.349,E2 -1694.349} C_VEL
LIN {X 0,Y 580.984,Z 320.876,A -85,B 0,C 180,E1 -1694.454,E2 -1694.454} C_VEL
LIN {X 0,Y 580.813,Z 424.873,A -85,B 0,C 180,E1 -1695.762,E2 -1695.762} C_VEL
LIN {X 0,Y 580.739,Z 438.436,A -85,B 0,C 180,E1 -1696.083,E2 -1696.083} C_VEL
LIN {X 0,Y 580.685,Z 451.031,A -85,B 0,C 180,E1 -1696.528,E2 -1696.528} C_VEL
LIN {X 0,Y 580.538,Z 462.224,A -85,B 0,C 180,E1 -1697.058,E2 -1697.058} C_VEL
LIN {X 0,Y 580.471,Z 473.85,A -85,B 0,C 180,E1 -1697.768,E2 -1697.768} C_VEL
LIN {X 0,Y 580.351,Z 484.387,A -85,B 0,C 180,E1 -1698.572,E2 -1698.572} C_VEL
LIN {X 0,Y 580.286,Z 494.474,A -85,B 0,C 180,E1 -1699.533,E2 -1699.533} C_VEL
LIN {X 0,Y 580.188,Z 503.387,A -85,B 0,C 180,E1 -1700.588,E2 -1700.588} C_VEL
LIN {X 0,Y 580.141,Z 510.531,A -85,B 0,C 180,E1 -1701.641,E2 -1701.641} C_VEL
LIN {X 0,Y 580.126,Z 516.218,A -85,B 0,C 180,E1 -1702.692,E2 -1702.692} C_VEL
LIN {X 0,Y 580.084,Z 520.692,A -85,B 0,C 180,E1 -1703.74,E2 -1703.74} C_VEL
LIN {X 0,Y 580.113,Z 523.051,A -85,B 0,C 180,E1 -1704.438,E2 -1704.438} C_VEL
LIN {X 0,Y 580.035,Z 524.977,A -85,B 0,C 180,E1 -1705.135,E2 -1705.135} C_VEL
LIN {X 0,Y 580.089,Z 526.483,A -85,B 0,C 180,E1 -1705.831,E2 -1705.831} C_VEL
LIN {X 0,Y 580.107,Z 527.538,A -85,B 0,C 180,E1 -1706.527,E2 -1706.527} C_VEL
LIN {X 0,Y 580.039,Z 528.477,A -85,B 0,C 180,E1 -1707.917,E2 -1707.917} C_VEL
LIN {X 0,Y 580.046,Z 528.368,A -85,B 0,C 180,E1 -1708.611,E2 -1708.611} C_VEL
LIN {X 0,Y 580.04,Z 526.907,A -85,B 0,C 180,E1 -1710,E2 -1710} C_VEL
LIN {X 0,Y 580.041,Z 525.588,A -85,B 0,C 180,E1 -1710.694,E2 -1710.694} C_VEL
LIN {X 0,Y 580.085,Z 522.795,A -85,B 0,C 180,E1 -1711.736,E2 -1711.736} C_VEL
LIN {X 0,Y 580.066,Z 518.99,A -85,B 0,C 180,E1 -1712.778,E2 -1712.778} C_VEL
LIN {X 0,Y 580.141,Z 514.069,A -85,B 0,C 180,E1 -1713.82,E2 -1713.82} C_VEL
LIN {X 0,Y 580.206,Z 507.886,A -85,B 0,C 180,E1 -1714.864,E2 -1714.864} C_VEL
LIN {X 0,Y 580.209,Z 500.19,A -85,B 0,C 180,E1 -1715.909,E2 -1715.909} C_VEL
LIN {X 0,Y 580.288,Z 491.861,A -85,B 0,C 180,E1 -1716.827,E2 -1716.827} C_VEL
LIN {X 0,Y 580.369,Z 481.675,A -85,B 0,C 180,E1 -1717.742,E2 -1717.742} C_VEL
LIN {X 0,Y 580.498,Z 470.759,A -85,B 0,C 180,E1 -1718.529,E2 -1718.529} C_VEL
LIN {X 0,Y 580.62,Z 460.087,A -85,B 0,C 180,E1 -1719.141,E2 -1719.141} C_VEL
LIN {X 0,Y 580.686,Z 448.38,A -85,B 0,C 180,E1 -1719.667,E2 -1719.667} C_VEL
LIN {X 0,Y 580.764,Z 435.787,A -85,B 0,C 180,E1 -1720.084,E2 -1720.084} C_VEL
LIN {X 0,Y 580.798,Z 423.883,A -85,B 0,C 180,E1 -1720.347,E2 -1720.347} C_VEL
LIN {X 0,Y 580.856,Z 318.761,A -85,B 0,C 180,E1 -1721.666,E2 -1721.666} C_VEL
LIN {X 0,Y 580.468,Z 315.679,A -85,B 0,C 180,E1 -1721.748,E2 -1721.748} C_VEL
LIN {X 0,Y 580.6,Z 294.296,A -85,B 0,C 180,E1 -1724.511,E2 -1724.511} C_VEL
LIN {X 0,Y 580.79,Z 270.837,A -85,B 0,C 180,E1 -1727.609,E2 -1727.609} C_VEL
LIN {X 0,Y 580.972,Z 250.418,A -85,B 0,C 180,E1 -1730.352,E2 -1730.352} C_VEL
LIN {X 0,Y 581.048,Z 239.52,A -85,B 0,C 180,E1 -1731.834,E2 -1731.834} C_VEL
LIN {X 0,Y 580.313,Z 235.927,A -85,B 0,C 180,E1 -1732.402,E2 -1732.402} C_VEL
LIN {X 0,Y 580.31,Z 235.816,A -85,B 0,C 180,E1 -1735.079,E2 -1735.079} C_VEL
LIN {X 0,Y 580.299,Z 235.822,A -85,B 0,C 180,E1 -1738.185,E2 -1738.185} C_VEL
LIN {X 0,Y 580.285,Z 235.822,A -85,B 0,C 180,E1 -1740.693,E2 -1740.693} C_VEL
LIN {X 0,Y 580.306,Z 235.826,A -85,B 0,C 180,E1 -1743.316,E2 -1743.316} C_VEL
LIN {X 0,Y 580.246,Z 235.831,A -85,B 0,C 180,E1 -1745.755,E2 -1745.755} C_VEL
LIN {X 0,Y 580.285,Z 235.822,A -85,B 0,C 180,E1 -1748.146,E2 -1748.146} C_VEL
LIN {X 0,Y 580.297,Z 235.823,A -85,B 0,C 180,E1 -1750.843,E2 -1750.843} C_VEL
LIN {X 0,Y 580.288,Z 235.824,A -85,B 0,C 180,E1 -1753.656,E2 -1753.656} C_VEL
LIN {X 0,Y 580.274,Z 235.824,A -85,B 0,C 180,E1 -1756.609,E2 -1756.609} C_VEL
LIN {X 0,Y 580.297,Z 235.828,A -85,B 0,C 180,E1 -1759.156,E2 -1759.156} C_VEL
LIN {X 0,Y 580.288,Z 235.821,A -85,B 0,C 180,E1 -1761.926,E2 -1761.926} C_VEL
LIN {X 0,Y 580.303,Z 235.821,A -85,B 0,C 180,E1 -1764.456,E2 -1764.456} C_VEL
LIN {X 0,Y 580.286,Z 235.828,A -85,B 0,C 180,E1 -1766.974,E2 -1766.974} C_VEL
LIN {X 0,Y 580.306,Z 235.822,A -85,B 0,C 180,E1 -1769.425,E2 -1769.425} C_VEL
LIN {X 0,Y 580.294,Z 235.82,A -85,B 0,C 180,E1 -1772.14,E2 -1772.14} C_VEL
LIN {X 0,Y 580.316,Z 235.82,A -85,B 0,C 180,E1 -1775.269,E2 -1775.269} C_VEL
LIN {X 0,Y 580.269,Z 235.824,A -85,B 0,C 180,E1 -1777.947,E2 -1777.947} C_VEL
LIN {X 0,Y 580.312,Z 235.826,A -85,B 0,C 180,E1 -1780.914,E2 -1780.914} C_VEL
LIN {X 0,Y 580.276,Z 235.822,A -85,B 0,C 180,E1 -1783.825,E2 -1783.825} C_VEL
LIN {X 0,Y 580.32,Z 235.817,A -85,B 0,C 180,E1 -1785.983,E2 -1785.983} C_VEL
LIN {X 0,Y 580.297,Z 235.826,A -85,B 0,C 180,E1 -1788.826,E2 -1788.826} C_VEL
LIN {X 0,Y 580.327,Z 235.816,A -85,B 0,C 180,E1 -1791.644,E2 -1791.644} C_VEL
LIN {X 0,Y 580.32,Z 235.825,A -85,B 0,C 180,E1 -1794.44,E2 -1794.44} C_VEL
LIN {X 0,Y 580.339,Z 235.816,A -85,B 0,C 180,E1 -1797.223,E2 -1797.223} C_VEL
LIN {X 0,Y 580.345,Z 235.817,A -85,B 0,C 180,E1 -1800,E2 -1800} C_VEL
LIN {X 0,Y 580.337,Z 235.819,A -85,B 0,C 180,E1 -1802.776,E2 -1802.776} C_VEL
LIN {X 0,Y 580.32,Z 235.816,A -85,B 0,C 180,E1 -1805.56,E2 -1805.56} C_VEL
LIN {X 0,Y 580.328,Z 235.826,A -85,B 0,C 180,E1 -1808.356,E2 -1808.356} C_VEL
LIN {X 0,Y 580.291,Z 235.82,A -85,B 0,C 180,E1 -1811.191,E2 -1811.191} C_VEL
LIN {X 0,Y 580.32,Z 235.824,A -85,B 0,C 180,E1 -1814.017,E2 -1814.017} C_VEL
LIN {X 0,Y 580.306,Z 235.819,A -85,B 0,C 180,E1 -1816.915,E2 -1816.915} C_VEL
LIN {X 0,Y 580.3,Z 235.824,A -85,B 0,C 180,E1 -1819.822,E2 -1819.822} C_VEL
LIN {X 0,Y 580.288,Z 235.822,A -85,B 0,C 180,E1 -1822.803,E2 -1822.803} C_VEL
LIN {X 0,Y 580.3,Z 235.819,A -85,B 0,C 180,E1 -1825.08,E2 -1825.08} C_VEL
LIN {X 0,Y 580.295,Z 235.826,A -85,B 0,C 180,E1 -1828.186,E2 -1828.186} C_VEL
LIN {X 0,Y 580.293,Z 235.819,A -85,B 0,C 180,E1 -1830.698,E2 -1830.698} C_VEL
LIN {X 0,Y 580.298,Z 235.822,A -85,B 0,C 180,E1 -1833.317,E2 -1833.317} C_VEL
LIN {X 0,Y 580.321,Z 235.825,A -85,B 0,C 180,E1 -1835.768,E2 -1835.768} C_VEL
LIN {X 0,Y 580.284,Z 235.827,A -85,B 0,C 180,E1 -1838.147,E2 -1838.147} C_VEL
LIN {X 0,Y 580.295,Z 235.82,A -85,B 0,C 180,E1 -1840.844,E2 -1840.844} C_VEL
LIN {X 0,Y 580.274,Z 235.831,A -85,B 0,C 180,E1 -1843.658,E2 -1843.658} C_VEL
LIN {X 0,Y 580.283,Z 235.82,A -85,B 0,C 180,E1 -1846.609,E2 -1846.609} C_VEL
LIN {X 0,Y 580.296,Z 235.818,A -85,B 0,C 180,E1 -1849.157,E2 -1849.157} C_VEL
LIN {X 0,Y 580.287,Z 235.826,A -85,B 0,C 180,E1 -1851.928,E2 -1851.928} C_VEL
LIN {X 0,Y 580.25,Z 235.824,A -85,B 0,C 180,E1 -1854.453,E2 -1854.453} C_VEL
LIN {X 0,Y 580.291,Z 235.823,A -85,B 0,C 180,E1 -1856.976,E2 -1856.976} C_VEL
LIN {X 0,Y 580.294,Z 235.828,A -85,B 0,C 180,E1 -1859.426,E2 -1859.426} C_VEL
LIN {X 0,Y 580.297,Z 235.823,A -85,B 0,C 180,E1 -1862.142,E2 -1862.142} C_VEL
LIN {X 0,Y 580.321,Z 235.827,A -85,B 0,C 180,E1 -1865.27,E2 -1865.27} C_VEL
LIN {X 0,Y 580.359,Z 236.038,A -85,B 0,C 180,E1 -1866.584,E2 -1866.584} C_VEL
LIN {X 0,Y 581.248,Z 241.117,A -85,B 0,C 180,E1 -1867.238,E2 -1867.238} C_VEL
LIN {X 0,Y 580.973,Z 266.537,A -85,B 0,C 180,E1 -1870.202,E2 -1870.202} C_VEL
LIN {X 0,Y 580.674,Z 291.956,A -85,B 0,C 180,E1 -1873.114,E2 -1873.114} C_VEL
LIN {X 0,Y 580.706,Z 295.038,A -85,B 0,C 180,E1 -1873.432,E2 -1873.432} C_VEL
LIN {X 0,Y 581.393,Z 299.642,A -85,B 0,C 180,E1 -1873.519,E2 -1873.519} C_VEL
LIN {X 0,Y 581.146,Z 433.9,A -85,B 0,C 180,E1 -1875.221,E2 -1875.221} C_VEL
LIN {X 0,Y 581.061,Z 447.881,A -85,B 0,C 180,E1 -1875.54,E2 -1875.54} C_VEL
LIN {X 0,Y 580.914,Z 461.718,A -85,B 0,C 180,E1 -1875.998,E2 -1875.998} C_VEL
LIN {X 0,Y 580.791,Z 475.647,A -85,B 0,C 180,E1 -1876.619,E2 -1876.619} C_VEL
LIN {X 0,Y 580.656,Z 488.104,A -85,B 0,C 180,E1 -1877.328,E2 -1877.328} C_VEL
LIN {X 0,Y 580.524,Z 500.644,A -85,B 0,C 180,E1 -1878.212,E2 -1878.212} C_VEL
LIN {X 0,Y 580.441,Z 511.893,A -85,B 0,C 180,E1 -1879.189,E2 -1879.189} C_VEL
LIN {X 0,Y 580.276,Z 521.853,A -85,B 0,C 180,E1 -1880.238,E2 -1880.238} C_VEL
LIN {X 0,Y 580.241,Z 530.173,A -85,B 0,C 180,E1 -1881.292,E2 -1881.292} C_VEL
LIN {X 0,Y 580.165,Z 538.128,A -85,B 0,C 180,E1 -1882.518,E2 -1882.518} C_VEL
LIN {X 0,Y 580.103,Z 544.528,A -85,B 0,C 180,E1 -1883.74,E2 -1883.74} C_VEL
LIN {X 0,Y 580.078,Z 548.962,A -85,B 0,C 180,E1 -1884.787,E2 -1884.787} C_VEL
LIN {X 0,Y 580.102,Z 552.443,A -85,B 0,C 180,E1 -1885.832,E2 -1885.832} C_VEL
LIN {X 0,Y 580.041,Z 555.832,A -85,B 0,C 180,E1 -1887.222,E2 -1887.222} C_VEL
LIN {X 0,Y 580.041,Z 557.832,A -85,B 0,C 180,E1 -1888.611,E2 -1888.611} C_VEL
LIN {X 0,Y 580.036,Z 558.5,A -85,B 0,C 180,E1 -1890,E2 -1890} C_VEL
LIN {X 0,Y 580.041,Z 557.833,A -85,B 0,C 180,E1 -1891.389,E2 -1891.389} C_VEL
LIN {X 0,Y 580.041,Z 555.833,A -85,B 0,C 180,E1 -1892.778,E2 -1892.778} C_VEL
LIN {X 0,Y 580.102,Z 552.444,A -85,B 0,C 180,E1 -1894.169,E2 -1894.169} C_VEL
LIN {X 0,Y 580.128,Z 547.568,A -85,B 0,C 180,E1 -1895.562,E2 -1895.562} C_VEL
LIN {X 0,Y 580.141,Z 541.053,A -85,B 0,C 180,E1 -1896.958,E2 -1896.958} C_VEL
LIN {X 0,Y 580.192,Z 533.801,A -85,B 0,C 180,E1 -1898.183,E2 -1898.183} C_VEL
LIN {X 0,Y 580.283,Z 524.824,A -85,B 0,C 180,E1 -1899.41,E2 -1899.41} C_VEL
LIN {X 0,Y 580.356,Z 515.393,A -85,B 0,C 180,E1 -1900.466,E2 -1900.466} C_VEL
LIN {X 0,Y 580.475,Z 505.322,A -85,B 0,C 180,E1 -1901.404,E2 -1901.404} C_VEL
LIN {X 0,Y 580.617,Z 493.435,A -85,B 0,C 180,E1 -1902.318,E2 -1902.318} C_VEL
LIN {X 0,Y 580.73,Z 480.649,A -85,B 0,C 180,E1 -1903.115,E2 -1903.115} C_VEL
LIN {X 0,Y 580.897,Z 468.16,A -85,B 0,C 180,E1 -1903.735,E2 -1903.735} C_VEL
LIN {X 0,Y 581.023,Z 455.01,A -85,B 0,C 180,E1 -1904.242,E2 -1904.242} C_VEL
LIN {X 0,Y 581.112,Z 441.914,A -85,B 0,C 180,E1 -1904.612,E2 -1904.612} C_VEL
LIN {X 0,Y 581.163,Z 428.136,A -85,B 0,C 180,E1 -1904.868,E2 -1904.868} C_VEL
LIN {X 0,Y 581.321,Z 298.629,A -85,B 0,C 180,E1 -1906.495,E2 -1906.495} C_VEL
LIN {X 0,Y 580.674,Z 294.679,A -85,B 0,C 180,E1 -1906.592,E2 -1906.592} C_VEL
LIN {X 0,Y 580.92,Z 269.226,A -85,B 0,C 180,E1 -1909.489,E2 -1909.489} C_VEL
LIN {X 0,Y 581.238,Z 242.705,A -85,B 0,C 180,E1 -1912.575,E2 -1912.575} C_VEL
LIN {X 0,Y 580.812,Z 238.175,A -85,B 0,C 180,E1 -1913.129,E2 -1913.129} C_VEL
LIN {X 0,Y 580.322,Z 235.915,A -85,B 0,C 180,E1 -1913.452,E2 -1913.452} C_VEL
LIN {X 0,Y 580.293,Z 235.823,A -85,B 0,C 180,E1 -1915.848,E2 -1915.848} C_VEL
LIN {X 0,Y 580.299,Z 235.826,A -85,B 0,C 180,E1 -1918.185,E2 -1918.185} C_VEL
LIN {X 0,Y 580.282,Z 235.828,A -85,B 0,C 180,E1 -1920.694,E2 -1920.694} C_VEL
LIN {X 0,Y 580.304,Z 235.82,A -85,B 0,C 180,E1 -1923.316,E2 -1923.316} C_VEL
LIN {X 0,Y 580.244,Z 235.827,A -85,B 0,C 180,E1 -1925.756,E2 -1925.756} C_VEL
LIN {X 0,Y 580.285,Z 235.826,A -85,B 0,C 180,E1 -1928.146,E2 -1928.146} C_VEL
LIN {X 0,Y 580.296,Z 235.822,A -85,B 0,C 180,E1 -1930.843,E2 -1930.843} C_VEL
LIN {X 0,Y 580.285,Z 235.823,A -85,B 0,C 180,E1 -1933.656,E2 -1933.656} C_VEL
LIN {X 0,Y 580.272,Z 235.827,A -85,B 0,C 180,E1 -1936.609,E2 -1936.609} C_VEL
LIN {X 0,Y 580.296,Z 235.819,A -85,B 0,C 180,E1 -1939.156,E2 -1939.156} C_VEL
LIN {X 0,Y 580.286,Z 235.828,A -85,B 0,C 180,E1 -1941.926,E2 -1941.926} C_VEL
LIN {X 0,Y 580.302,Z 235.823,A -85,B 0,C 180,E1 -1944.456,E2 -1944.456} C_VEL
LIN {X 0,Y 580.285,Z 235.822,A -85,B 0,C 180,E1 -1946.975,E2 -1946.975} C_VEL
LIN {X 0,Y 580.304,Z 235.819,A -85,B 0,C 180,E1 -1949.426,E2 -1949.426} C_VEL
LIN {X 0,Y 580.313,Z 235.826,A -85,B 0,C 180,E1 -1952.137,E2 -1952.137} C_VEL
LIN {X 0,Y 580.315,Z 235.818,A -85,B 0,C 180,E1 -1955.269,E2 -1955.269} C_VEL
LIN {X 0,Y 580.269,Z 235.833,A -85,B 0,C 180,E1 -1957.947,E2 -1957.947} C_VEL
LIN {X 0,Y 580.311,Z 235.818,A -85,B 0,C 180,E1 -1960.914,E2 -1960.914} C_VEL
LIN {X 0,Y 580.277,Z 235.832,A -85,B 0,C 180,E1 -1963.826,E2 -1963.826} C_VEL
LIN {X 0,Y 580.321,Z 235.823,A -85,B 0,C 180,E1 -1965.983,E2 -1965.983} C_VEL
LIN {X 0,Y 580.297,Z 235.819,A -85,B 0,C 180,E1 -1968.827,E2 -1968.827} C_VEL
LIN {X 0,Y 580.328,Z 235.826,A -85,B 0,C 180,E1 -1971.644,E2 -1971.644} C_VEL
LIN {X 0,Y 580.32,Z 235.817,A -85,B 0,C 180,E1 -1974.44,E2 -1974.44} C_VEL
LIN {X 0,Y 580.337,Z 235.819,A -85,B 0,C 180,E1 -1977.224,E2 -1977.224} C_VEL
LIN {X 0,Y 580.345,Z 235.817,A -85,B 0,C 180,E1 -1980,E2 -1980} C_VEL
LIN {X 0,Y 580.339,Z 235.815,A -85,B 0,C 180,E1 -1982.777,E2 -1982.777} C_VEL
LIN {X 0,Y 580.319,Z 235.825,A -85,B 0,C 180,E1 -1985.56,E2 -1985.56} C_VEL
LIN {X 0,Y 580.328,Z 235.816,A -85,B 0,C 180,E1 -1988.356,E2 -1988.356} C_VEL
LIN {X 0,Y 580.293,Z 235.828,A -85,B 0,C 180,E1 -1991.192,E2 -1991.192} C_VEL
LIN {X 0,Y 580.321,Z 235.818,A -85,B 0,C 180,E1 -1994.017,E2 -1994.017} C_VEL
LIN {X 0,Y 580.307,Z 235.822,A -85,B 0,C 180,E1 -1996.915,E2 -1996.915} C_VEL
LIN {X 0,Y 580.302,Z 235.82,A -85,B 0,C 180,E1 -1999.823,E2 -1999.823} C_VEL
LIN {X 0,Y 580.277,Z 235.83,A -85,B 0,C 180,E1 -2001.338,E2 -2001.338} C_VEL
LIN {X 0,Y 579.582,Z 235.912,A -85,B 0,C 180,E1 -2001.917,E2 -2001.917} C_VEL
LIN {X 0,Y 576.706,Z 236.272,A -85,B 0,C 180,E1 -2002.857,E2 -2002.857} C_VEL
LIN {X 0,Y 574.312,Z 236.568,A -85,B 0,C 180,E1 -2003.613,E2 -2003.613} C_VEL
LIN {X 0,Y 573.313,Z 236.69,A -85,B 0,C 180,E1 -2004.197,E2 -2004.197} C_VEL
LIN {X 0,Y 573.246,Z 236.698,A -85,B 0,C 180,E1 -2004.394,E2 -2004.394} C_VEL
LIN {X 0,Y 573.247,Z 236.706,A -85,B 0,C 180,E1 -2006.977,E2 -2006.977} C_VEL
LIN {X 0,Y 573.243,Z 236.701,A -85,B 0,C 180,E1 -2009.489,E2 -2009.489} C_VEL
LIN {X 0,Y 573.251,Z 236.699,A -85,B 0,C 180,E1 -2012.23,E2 -2012.23} C_VEL
LIN {X 0,Y 573.248,Z 236.704,A -85,B 0,C 180,E1 -2014.774,E2 -2014.774} C_VEL
LIN {X 0,Y 573.252,Z 236.704,A -85,B 0,C 180,E1 -2017.167,E2 -2017.167} C_VEL
LIN {X 0,Y 573.246,Z 236.697,A -85,B 0,C 180,E1 -2019.608,E2 -2019.608} C_VEL
LIN {X 0,Y 573.238,Z 236.706,A -85,B 0,C 180,E1 -2022.642,E2 -2022.642} C_VEL
LIN {X 0,Y 573.239,Z 236.7,A -85,B 0,C 180,E1 -2025.668,E2 -2025.668} C_VEL
LIN {X 0,Y 573.244,Z 236.704,A -85,B 0,C 180,E1 -2028.545,E2 -2028.545} C_VEL
LIN {X 0,Y 573.242,Z 236.696,A -85,B 0,C 180,E1 -2031.299,E2 -2031.299} C_VEL
LIN {X 0,Y 573.214,Z 236.704,A -85,B 0,C 180,E1 -2034.019,E2 -2034.019} C_VEL
LIN {X 0,Y 573.24,Z 236.704,A -85,B 0,C 180,E1 -2036.517,E2 -2036.517} C_VEL
LIN {X 0,Y 573.226,Z 236.704,A -85,B 0,C 180,E1 -2039.119,E2 -2039.119} C_VEL
LIN {X 0,Y 573.238,Z 236.699,A -85,B 0,C 180,E1 -2041.436,E2 -2041.436} C_VEL
LIN {X 0,Y 573.298,Z 236.919,A -85,B 0,C 180,E1 -2043.541,E2 -2043.541} C_VEL
LIN {X 0,Y 574.264,Z 242.996,A -85,B 0,C 180,E1 -2044.444,E2 -2044.444} C_VEL
LIN {X 0,Y 573.948,Z 264.006,A -85,B 0,C 180,E1 -2047.312,E2 -2047.312} C_VEL
LIN {X 0,Y 573.738,Z 282.147,A -85,B 0,C 180,E1 -2049.755,E2 -2049.755} C_VEL
LIN {X 0,Y 573.523,Z 304.43,A -85,B 0,C 180,E1 -2052.713,E2 -2052.713} C_VEL
LIN {X 0,Y 573.449,Z 315.748,A -85,B 0,C 180,E1 -2054.176,E2 -2054.176} C_VEL
LIN {X 0,Y 574.083,Z 320.689,A -85,B 0,C 180,E1 -2054.285,E2 -2054.285} C_VEL
LIN {X 0,Y 573.885,Z 425.136,A -85,B 0,C 180,E1 -2055.616,E2 -2055.616} C_VEL
LIN {X 0,Y 573.803,Z 438.36,A -85,B 0,C 180,E1 -2055.934,E2 -2055.934} C_VEL
LIN {X 0,Y 573.74,Z 450.414,A -85,B 0,C 180,E1 -2056.361,E2 -2056.361} C_VEL
LIN {X 0,Y 573.585,Z 461.78,A -85,B 0,C 180,E1 -2056.899,E2 -2056.899} C_VEL
LIN {X 0,Y 573.454,Z 473.488,A -85,B 0,C 180,E1 -2057.616,E2 -2057.616} C_VEL
LIN {X 0,Y 573.337,Z 483.984,A -85,B 0,C 180,E1 -2058.421,E2 -2058.421} C_VEL
LIN {X 0,Y 573.258,Z 492.891,A -85,B 0,C 180,E1 -2059.258,E2 -2059.258} C_VEL
LIN {X 0,Y 573.13,Z 501.837,A -85,B 0,C 180,E1 -2060.293,E2 -2060.293} C_VEL
LIN {X 0,Y 573.103,Z 509.273,A -85,B 0,C 180,E1 -2061.36,E2 -2061.36} C_VEL
LIN {X 0,Y 573.046,Z 516.107,A -85,B 0,C 180,E1 -2062.601,E2 -2062.601} C_VEL
LIN {X 0,Y 573.011,Z 520.606,A -85,B 0,C 180,E1 -2063.663,E2 -2063.663} C_VEL
LIN {X 0,Y 573.036,Z 522.978,A -85,B 0,C 180,E1 -2064.369,E2 -2064.369} C_VEL
LIN {X 0,Y 572.944,Z 524.916,A -85,B 0,C 180,E1 -2065.074,E2 -2065.074} C_VEL
LIN {X 0,Y 573.009,Z 526.439,A -85,B 0,C 180,E1 -2065.78,E2 -2065.78} C_VEL
LIN {X 0,Y 573.007,Z 527.51,A -85,B 0,C 180,E1 -2066.484,E2 -2066.484} C_VEL
LIN {X 0,Y 572.938,Z 528.472,A -85,B 0,C 180,E1 -2067.891,E2 -2067.891} C_VEL
LIN {X 0,Y 572.946,Z 528.379,A -85,B 0,C 180,E1 -2068.594,E2 -2068.594} C_VEL
LIN {X 0,Y 572.941,Z 526.946,A -85,B 0,C 180,E1 -2070,E2 -2070} C_VEL
LIN {X 0,Y 572.942,Z 525.638,A -85,B 0,C 180,E1 -2070.703,E2 -2070.703} C_VEL
LIN {X 0,Y 572.994,Z 522.868,A -85,B 0,C 180,E1 -2071.757,E2 -2071.757} C_VEL
LIN {X 0,Y 572.983,Z 519.088,A -85,B 0,C 180,E1 -2072.812,E2 -2072.812} C_VEL
LIN {X 0,Y 573.071,Z 514.194,A -85,B 0,C 180,E1 -2073.867,E2 -2073.867} C_VEL
LIN {X 0,Y 573.125,Z 508.041,A -85,B 0,C 180,E1 -2074.924,E2 -2074.924} C_VEL
LIN {X 0,Y 573.158,Z 500.392,A -85,B 0,C 180,E1 -2075.982,E2 -2075.982} C_VEL
LIN {X 0,Y 573.248,Z 492.265,A -85,B 0,C 180,E1 -2076.895,E2 -2076.895} C_VEL
LIN {X 0,Y 573.358,Z 481.968,A -85,B 0,C 180,E1 -2077.837,E2 -2077.837} C_VEL
LIN {X 0,Y 573.506,Z 471.147,A -85,B 0,C 180,E1 -2078.634,E2 -2078.634} C_VEL
LIN {X 0,Y 573.64,Z 460.57,A -85,B 0,C 180,E1 -2079.253,E2 -2079.253} C_VEL
LIN {X 0,Y 573.739,Z 448.998,A -85,B 0,C 180,E1 -2079.785,E2 -2079.785} C_VEL
LIN {X 0,Y 573.814,Z 435.865,A -85,B 0,C 180,E1 -2080.229,E2 -2080.229} C_VEL
LIN {X 0,Y 573.861,Z 424.015,A -85,B 0,C 180,E1 -2080.496,E2 -2080.496} C_VEL
LIN {X 0,Y 573.996,Z 319.746,A -85,B 0,C 180,E1 -2081.819,E2 -2081.819} C_VEL
LIN {X 0,Y 573.457,Z 315.766,A -85,B 0,C 180,E1 -2081.912,E2 -2081.912} C_VEL
LIN {X 0,Y 573.628,Z 294.763,A -85,B 0,C 180,E1 -2084.655,E2 -2084.655} C_VEL
LIN {X 0,Y 573.873,Z 271.032,A -85,B 0,C 180,E1 -2087.828,E2 -2087.828} C_VEL
LIN {X 0,Y 574.108,Z 250.582,A -85,B 0,C 180,E1 -2090.606,E2 -2090.606} C_VEL
LIN {X 0,Y 574.166,Z 241.044,A -85,B 0,C 180,E1 -2091.921,E2 -2091.921} C_VEL
LIN {X 0,Y 573.267,Z 236.838,A -85,B 0,C 180,E1 -2092.574,E2 -2092.574} C_VEL
LIN {X 0,Y 573.257,Z 236.692,A -85,B 0,C 180,E1 -2095.409,E2 -2095.409} C_VEL
LIN {X 0,Y 573.239,Z 236.701,A -85,B 0,C 180,E1 -2098.564,E2 -2098.564} C_VEL
LIN {X 0,Y 573.227,Z 236.703,A -85,B 0,C 180,E1 -2100.993,E2 -2100.993} C_VEL
LIN {X 0,Y 573.264,Z 236.701,A -85,B 0,C 180,E1 -2103.523,E2 -2103.523} C_VEL
LIN {X 0,Y 573.215,Z 236.704,A -85,B 0,C 180,E1 -2106.051,E2 -2106.051} C_VEL
LIN {X 0,Y 573.239,Z 236.701,A -85,B 0,C 180,E1 -2108.701,E2 -2108.701} C_VEL
LIN {X 0,Y 573.253,Z 236.702,A -85,B 0,C 180,E1 -2111.595,E2 -2111.595} C_VEL
LIN {X 0,Y 573.239,Z 236.699,A -85,B 0,C 180,E1 -2114.332,E2 -2114.332} C_VEL
LIN {X 0,Y 573.238,Z 236.706,A -85,B 0,C 180,E1 -2117.358,E2 -2117.358} C_VEL
LIN {X 0,Y 573.246,Z 236.696,A -85,B 0,C 180,E1 -2120.392,E2 -2120.392} C_VEL
LIN {X 0,Y 573.254,Z 236.708,A -85,B 0,C 180,E1 -2123.077,E2 -2123.077} C_VEL
LIN {X 0,Y 573.269,Z 236.694,A -85,B 0,C 180,E1 -2125.671,E2 -2125.671} C_VEL
LIN {X 0,Y 573.244,Z 236.698,A -85,B 0,C 180,E1 -2128.184,E2 -2128.184} C_VEL
LIN {X 0,Y 573.264,Z 236.701,A -85,B 0,C 180,E1 -2130.634,E2 -2130.634} C_VEL
LIN {X 0,Y 573.235,Z 236.702,A -85,B 0,C 180,E1 -2133.506,E2 -2133.506} C_VEL
LIN {X 0,Y 573.228,Z 236.7,A -85,B 0,C 180,E1 -2136.134,E2 -2136.134} C_VEL
LIN {X 0,Y 573.245,Z 236.702,A -85,B 0,C 180,E1 -2139.173,E2 -2139.173} C_VEL
LIN {X 0,Y 573.231,Z 236.701,A -85,B 0,C 180,E1 -2141.411,E2 -2141.411} C_VEL
LIN {X 0,Y 573.252,Z 236.697,A -85,B 0,C 180,E1 -2143.621,E2 -2143.621} C_VEL
LIN {X 0,Y 573.232,Z 236.706,A -85,B 0,C 180,E1 -2146.529,E2 -2146.529} C_VEL
LIN {X 0,Y 573.255,Z 236.705,A -85,B 0,C 180,E1 -2148.745,E2 -2148.745} C_VEL
LIN {X 0,Y 573.284,Z 236.693,A -85,B 0,C 180,E1 -2151.54,E2 -2151.54} C_VEL
LIN {X 0,Y 573.286,Z 236.7,A -85,B 0,C 180,E1 -2154.372,E2 -2154.372} C_VEL
LIN {X 0,Y 573.302,Z 236.693,A -85,B 0,C 180,E1 -2157.892,E2 -2157.892} C_VEL
LIN {X 0,Y 573.329,Z 236.693,A -85,B 0,C 180,E1 -2160.702,E2 -2160.702} C_VEL
LIN {X 0,Y 573.233,Z 236.7,A -85,B 0,C 180,E1 -2163.514,E2 -2163.514} C_VEL
LIN {X 0,Y 573.287,Z 236.693,A -85,B 0,C 180,E1 -2165.628,E2 -2165.628} C_VEL
LIN {X 0,Y 573.284,Z 236.702,A -85,B 0,C 180,E1 -2168.459,E2 -2168.459} C_VEL
LIN {X 0,Y 573.263,Z 236.695,A -85,B 0,C 180,E1 -2171.312,E2 -2171.312} C_VEL
LIN {X 0,Y 573.266,Z 236.705,A -85,B 0,C 180,E1 -2174.193,E2 -2174.193} C_VEL
LIN {X 0,Y 573.253,Z 236.697,A -85,B 0,C 180,E1 -2177.112,E2 -2177.112} C_VEL
LIN {X 0,Y 573.247,Z 236.707,A -85,B 0,C 180,E1 -2180.077,E2 -2180.077} C_VEL
LIN {X 0,Y 573.226,Z 236.701,A -85,B 0,C 180,E1 -2183.1,E2 -2183.1} C_VEL
LIN {X 0,Y 573.248,Z 236.699,A -85,B 0,C 180,E1 -2185.41,E2 -2185.41} C_VEL
LIN {X 0,Y 573.257,Z 236.706,A -85,B 0,C 180,E1 -2188.032,E2 -2188.032} C_VEL
LIN {X 0,Y 573.237,Z 236.697,A -85,B 0,C 180,E1 -2190.885,E2 -2190.885} C_VEL
LIN {X 0,Y 573.256,Z 236.701,A -85,B 0,C 180,E1 -2193.524,E2 -2193.524} C_VEL
LIN {X 0,Y 573.256,Z 236.702,A -85,B 0,C 180,E1 -2196.048,E2 -2196.048} C_VEL
LIN {X 0,Y 573.245,Z 236.699,A -85,B 0,C 180,E1 -2198.701,E2 -2198.701} C_VEL
LIN {X 0,Y 573.249,Z 236.705,A -85,B 0,C 180,E1 -2201.596,E2 -2201.596} C_VEL
LIN {X 0,Y 573.231,Z 236.702,A -85,B 0,C 180,E1 -2204.334,E2 -2204.334} C_VEL
LIN {X 0,Y 573.241,Z 236.701,A -85,B 0,C 180,E1 -2207.359,E2 -2207.359} C_VEL
LIN {X 0,Y 573.237,Z 236.7,A -85,B 0,C 180,E1 -2210.393,E2 -2210.393} C_VEL
LIN {X 0,Y 573.249,Z 236.7,A -85,B 0,C 180,E1 -2213.078,E2 -2213.078} C_VEL
LIN {X 0,Y 573.266,Z 236.705,A -85,B 0,C 180,E1 -2215.672,E2 -2215.672} C_VEL
LIN {X 0,Y 573.243,Z 236.697,A -85,B 0,C 180,E1 -2218.185,E2 -2218.185} C_VEL
LIN {X 0,Y 573.263,Z 236.698,A -85,B 0,C 180,E1 -2220.635,E2 -2220.635} C_VEL
LIN {X 0,Y 573.25,Z 236.703,A -85,B 0,C 180,E1 -2223.025,E2 -2223.025} C_VEL
LIN {X 0,Y 573.275,Z 236.703,A -85,B 0,C 180,E1 -2225.367,E2 -2225.367} C_VEL
LIN {X 0,Y 573.282,Z 236.905,A -85,B 0,C 180,E1 -2226.378,E2 -2226.378} C_VEL
LIN {X 0,Y 574.406,Z 242.72,A -85,B 0,C 180,E1 -2227.141,E2 -2227.141} C_VEL
LIN {X 0,Y 574.059,Z 268.219,A -85,B 0,C 180,E1 -2230.151,E2 -2230.151} C_VEL
LIN {X 0,Y 573.699,Z 293.545,A -85,B 0,C 180,E1 -2233.086,E2 -2233.086} C_VEL
LIN {X 0,Y 573.747,Z 295.04,A -85,B 0,C 180,E1 -2233.225,E2 -2233.225} C_VEL
LIN {X 0,Y 574.557,Z 299.64,A -85,B 0,C 180,E1 -2233.318,E2 -2233.318} C_VEL
LIN {X 0,Y 574.306,Z 432.654,A -85,B 0,C 180,E1 -2235.018,E2 -2235.018} C_VEL
LIN {X 0,Y 574.184,Z 446.898,A -85,B 0,C 180,E1 -2235.333,E2 -2235.333} C_VEL
LIN {X 0,Y 574.078,Z 460.311,A -85,B 0,C 180,E1 -2235.771,E2 -2235.771} C_VEL
LIN {X 0,Y 573.939,Z 473.883,A -85,B 0,C 180,E1 -2236.366,E2 -2236.366} C_VEL
LIN {X 0,Y 573.721,Z 486.684,A -85,B 0,C 180,E1 -2237.082,E2 -2237.082} C_VEL
LIN {X 0,Y 573.583,Z 498.318,A -85,B 0,C 180,E1 -2237.888,E2 -2237.888} C_VEL
LIN {X 0,Y 573.45,Z 509.455,A -85,B 0,C 180,E1 -2238.826,E2 -2238.826} C_VEL
LIN {X 0,Y 573.269,Z 520.335,A -85,B 0,C 180,E1 -2239.939,E2 -2239.939} C_VEL
LIN {X 0,Y 573.19,Z 528.913,A -85,B 0,C 180,E1 -2241.006,E2 -2241.006} C_VEL
LIN {X 0,Y 573.111,Z 537.117,A -85,B 0,C 180,E1 -2242.248,E2 -2242.248} C_VEL
LIN {X 0,Y 573.036,Z 543.448,A -85,B 0,C 180,E1 -2243.427,E2 -2243.427} C_VEL
LIN {X 0,Y 573.001,Z 548.961,A -85,B 0,C 180,E1 -2244.722,E2 -2244.722} C_VEL
LIN {X 0,Y 573.028,Z 552.443,A -85,B 0,C 180,E1 -2245.78,E2 -2245.78} C_VEL
LIN {X 0,Y 572.956,Z 555.832,A -85,B 0,C 180,E1 -2247.188,E2 -2247.188} C_VEL
LIN {X 0,Y 572.941,Z 557.833,A -85,B 0,C 180,E1 -2248.594,E2 -2248.594} C_VEL
LIN {X 0,Y 572.937,Z 558.5,A -85,B 0,C 180,E1 -2250,E2 -2250} C_VEL
LIN {X 0,Y 572.941,Z 557.833,A -85,B 0,C 180,E1 -2251.406,E2 -2251.406} C_VEL
LIN {X 0,Y 572.956,Z 555.834,A -85,B 0,C 180,E1 -2252.812,E2 -2252.812} C_VEL
LIN {X 0,Y 573.028,Z 552.445,A -85,B 0,C 180,E1 -2254.22,E2 -2254.22} C_VEL
LIN {X 0,Y 573.057,Z 547.568,A -85,B 0,C 180,E1 -2255.63,E2 -2255.63} C_VEL
LIN {X 0,Y 573.065,Z 542.818,A -85,B 0,C 180,E1 -2256.699,E2 -2256.699} C_VEL
LIN {X 0,Y 573.126,Z 536.038,A -85,B 0,C 180,E1 -2257.929,E2 -2257.929} C_VEL
LIN {X 0,Y 573.225,Z 527.559,A -85,B 0,C 180,E1 -2259.171,E2 -2259.171} C_VEL
LIN {X 0,Y 573.304,Z 518.708,A -85,B 0,C 180,E1 -2260.239,E2 -2260.239} C_VEL
